LIN {X 0,Y 247.812,Z 545.239,A -85,B 0,C 180,E1 -18999.797,E2 -18999.797} C_VEL
LIN {X 0,Y 248.949,Z 540.408,A -85,B 0,C 180,E1 -19003.052,E2 -19003.052} C_VEL
LIN {X 0,Y 250.872,Z 533.939,A -85,B 0,C 180,E1 -19006.268,E2 -19006.268} C_VEL
LIN {X 0,Y 252.75,Z 526.871,A -85,B 0,C 180,E1 -19009.018,E2 -19009.018} C_VEL
LIN {X 0,Y 254.982,Z 519.187,A -85,B 0,C 180,E1 -19011.42,E2 -19011.42} C_VEL
LIN {X 0,Y 257.581,Z 510.12,A -85,B 0,C 180,E1 -19013.731,E2 -19013.731} C_VEL
LIN {X 0,Y 260.595,Z 499.136,A -85,B 0,C 180,E1 -19015.991,E2 -19015.991} C_VEL
LIN {X 0,Y 263.396,Z 487.928,A -85,B 0,C 180,E1 -19017.835,E2 -19017.835} C_VEL
LIN {X 0,Y 266.028,Z 475.354,A -85,B 0,C 180,E1 -19019.498,E2 -19019.498} C_VEL
LIN {X 0,Y 268.183,Z 463.582,A -85,B 0,C 180,E1 -19020.731,E2 -19020.731} C_VEL
LIN {X 0,Y 270.195,Z 450.492,A -85,B 0,C 180,E1 -19021.783,E2 -19021.783} C_VEL
LIN {X 0,Y 271.759,Z 437.252,A -85,B 0,C 180,E1 -19022.563,E2 -19022.563} C_VEL
LIN {X 0,Y 272.875,Z 422.735,A -85,B 0,C 180,E1 -19023.129,E2 -19023.129} C_VEL
LIN {X 0,Y 275.889,Z 350.665,A -85,B 0,C 180,E1 -19024.953,E2 -19024.953} C_VEL
LIN {X 0,Y 276.102,Z 341.819,A -85,B 0,C 180,E1 -19025.198,E2 -19025.198} C_VEL
LIN {X 0,Y 269.628,Z 326.55,A -85,B 0,C 180,E1 -19026.671,E2 -19026.671} C_VEL
LIN {X 0,Y 261.498,Z 310.016,A -85,B 0,C 180,E1 -19028.578,E2 -19028.578} C_VEL
LIN {X 0,Y 254.853,Z 298.261,A -85,B 0,C 180,E1 -19030.206,E2 -19030.206} C_VEL
LIN {X 0,Y 249.821,Z 289.724,A -85,B 0,C 180,E1 -19031.561,E2 -19031.561} C_VEL
LIN {X 0,Y 249.021,Z 287.115,A -85,B 0,C 180,E1 -19032.795,E2 -19032.795} C_VEL
LIN {X 0,Y 249.016,Z 287.053,A -85,B 0,C 180,E1 -19037.362,E2 -19037.362} C_VEL
LIN {X 0,Y 249.035,Z 287.087,A -85,B 0,C 180,E1 -19041.621,E2 -19041.621} C_VEL
LIN {X 0,Y 249.058,Z 287.032,A -85,B 0,C 180,E1 -19045.641,E2 -19045.641} C_VEL
LIN {X 0,Y 249.048,Z 287.064,A -85,B 0,C 180,E1 -19049.472,E2 -19049.472} C_VEL
LIN {X 0,Y 249.07,Z 287.07,A -85,B 0,C 180,E1 -19053.162,E2 -19053.162} C_VEL
LIN {X 0,Y 249.075,Z 287.086,A -85,B 0,C 180,E1 -19056.732,E2 -19056.732} C_VEL
LIN {X 0,Y 249.105,Z 287.065,A -85,B 0,C 180,E1 -19060.211,E2 -19060.211} C_VEL
LIN {X 0,Y 249.238,Z 287.051,A -85,B 0,C 180,E1 -19063.621,E2 -19063.621} C_VEL
LIN {X 0,Y 249.239,Z 287.062,A -85,B 0,C 180,E1 -19068.616,E2 -19068.616} C_VEL
LIN {X 0,Y 249.449,Z 287.016,A -85,B 0,C 180,E1 -19071.902,E2 -19071.902} C_VEL
LIN {X 0,Y 249.32,Z 287.04,A -85,B 0,C 180,E1 -19075.745,E2 -19075.745} C_VEL
LIN {X 0,Y 248.758,Z 287.101,A -85,B 0,C 180,E1 -19077.097,E2 -19077.097} C_VEL
LIN {X 0,Y 246.053,Z 287.448,A -85,B 0,C 180,E1 -19079.305,E2 -19079.305} C_VEL
LIN {X 0,Y 242.805,Z 287.856,A -85,B 0,C 180,E1 -19082.025,E2 -19082.025} C_VEL
LIN {X 0,Y 242.407,Z 287.894,A -85,B 0,C 180,E1 -19082.966,E2 -19082.966} C_VEL
LIN {X 0,Y 242.428,Z 287.91,A -85,B 0,C 180,E1 -19086.659,E2 -19086.659} C_VEL
LIN {X 0,Y 242.309,Z 287.903,A -85,B 0,C 180,E1 -19090.022,E2 -19090.022} C_VEL
LIN {X 0,Y 242.151,Z 287.932,A -85,B 0,C 180,E1 -19095.142,E2 -19095.142} C_VEL
LIN {X 0,Y 242.066,Z 287.954,A -85,B 0,C 180,E1 -19098.625,E2 -19098.625} C_VEL
LIN {X 0,Y 242.008,Z 287.945,A -85,B 0,C 180,E1 -19102.18,E2 -19102.18} C_VEL
LIN {X 0,Y 242.063,Z 287.951,A -85,B 0,C 180,E1 -19105.838,E2 -19105.838} C_VEL
LIN {X 0,Y 242.026,Z 287.962,A -85,B 0,C 180,E1 -19109.581,E2 -19109.581} C_VEL
LIN {X 0,Y 241.977,Z 287.91,A -85,B 0,C 180,E1 -19113.493,E2 -19113.493} C_VEL
LIN {X 0,Y 241.983,Z 287.952,A -85,B 0,C 180,E1 -19117.583,E2 -19117.583} C_VEL
LIN {X 0,Y 241.94,Z 287.97,A -85,B 0,C 180,E1 -19121.922,E2 -19121.922} C_VEL
LIN {X 0,Y 241.976,Z 288.026,A -85,B 0,C 180,E1 -19124.674,E2 -19124.674} C_VEL
LIN {X 0,Y 243.43,Z 292.652,A -85,B 0,C 180,E1 -19127.066,E2 -19127.066} C_VEL
LIN {X 0,Y 245.542,Z 296.633,A -85,B 0,C 180,E1 -19127.779,E2 -19127.779} C_VEL
LIN {X 0,Y 251.81,Z 307.211,A -85,B 0,C 180,E1 -19129.449,E2 -19129.449} C_VEL
LIN {X 0,Y 259.928,Z 322.862,A -85,B 0,C 180,E1 -19131.503,E2 -19131.503} C_VEL
LIN {X 0,Y 267.648,Z 340.131,A -85,B 0,C 180,E1 -19133.371,E2 -19133.371} C_VEL
LIN {X 0,Y 270.071,Z 346.299,A -85,B 0,C 180,E1 -19133.951,E2 -19133.951} C_VEL
LIN {X 0,Y 270.223,Z 349.656,A -85,B 0,C 180,E1 -19134.082,E2 -19134.082} C_VEL
LIN {X 0,Y 266.583,Z 431,A -85,B 0,C 180,E1 -19136.193,E2 -19136.193} C_VEL
LIN {X 0,Y 265.194,Z 445.012,A -85,B 0,C 180,E1 -19136.811,E2 -19136.811} C_VEL
LIN {X 0,Y 263.479,Z 457.894,A -85,B 0,C 180,E1 -19137.647,E2 -19137.647} C_VEL
LIN {X 0,Y 261.144,Z 471.147,A -85,B 0,C 180,E1 -19138.798,E2 -19138.798} C_VEL
LIN {X 0,Y 258.544,Z 483.922,A -85,B 0,C 180,E1 -19140.259,E2 -19140.259} C_VEL
LIN {X 0,Y 255.96,Z 495.088,A -85,B 0,C 180,E1 -19141.867,E2 -19141.867} C_VEL
LIN {X 0,Y 253.272,Z 505.213,A -85,B 0,C 180,E1 -19143.643,E2 -19143.643} C_VEL
LIN {X 0,Y 250.226,Z 515.932,A -85,B 0,C 180,E1 -19145.968,E2 -19145.968} C_VEL
LIN {X 0,Y 247.534,Z 524.782,A -85,B 0,C 180,E1 -19148.341,E2 -19148.341} C_VEL
LIN {X 0,Y 245.329,Z 532.305,A -85,B 0,C 180,E1 -19150.827,E2 -19150.827} C_VEL
LIN {X 0,Y 243.603,Z 538.288,A -85,B 0,C 180,E1 -19153.232,E2 -19153.232} C_VEL
LIN {X 0,Y 242.131,Z 543.376,A -85,B 0,C 180,E1 -19155.717,E2 -19155.717} C_VEL
LIN {X 0,Y 240.791,Z 548.626,A -85,B 0,C 180,E1 -19159.064,E2 -19159.064} C_VEL
LIN {X 0,Y 240.204,Z 551.568,A -85,B 0,C 180,E1 -19161.588,E2 -19161.588} C_VEL
LIN {X 0,Y 239.8,Z 554.259,A -85,B 0,C 180,E1 -19164.956,E2 -19164.956} C_VEL
LIN {X 0,Y 239.768,Z 555.59,A -85,B 0,C 180,E1 -19168.32,E2 -19168.32} C_VEL
LIN {X 0,Y 239.802,Z 555.753,A -85,B 0,C 180,E1 -19170,E2 -19170} C_VEL
LIN {X 0,Y 239.727,Z 555.077,A -85,B 0,C 180,E1 -19173.361,E2 -19173.361} C_VEL
LIN {X 0,Y 239.955,Z 553.058,A -85,B 0,C 180,E1 -19176.728,E2 -19176.728} C_VEL
LIN {X 0,Y 240.584,Z 549.648,A -85,B 0,C 180,E1 -19180.094,E2 -19180.094} C_VEL
LIN {X 0,Y 241.671,Z 544.743,A -85,B 0,C 180,E1 -19183.453,E2 -19183.453} C_VEL
LIN {X 0,Y 243.115,Z 540.017,A -85,B 0,C 180,E1 -19185.94,E2 -19185.94} C_VEL
LIN {X 0,Y 244.834,Z 533.55,A -85,B 0,C 180,E1 -19188.689,E2 -19188.689} C_VEL
LIN {X 0,Y 247.121,Z 526.01,A -85,B 0,C 180,E1 -19191.26,E2 -19191.26} C_VEL
LIN {X 0,Y 249.716,Z 517.407,A -85,B 0,C 180,E1 -19193.643,E2 -19193.643} C_VEL
LIN {X 0,Y 252.713,Z 506.979,A -85,B 0,C 180,E1 -19195.976,E2 -19195.976} C_VEL
LIN {X 0,Y 255.58,Z 496.491,A -85,B 0,C 180,E1 -19197.87,E2 -19197.87} C_VEL
LIN {X 0,Y 258.224,Z 485.076,A -85,B 0,C 180,E1 -19199.557,E2 -19199.557} C_VEL
LIN {X 0,Y 260.813,Z 472.57,A -85,B 0,C 180,E1 -19201.02,E2 -19201.02} C_VEL
LIN {X 0,Y 263.278,Z 458.571,A -85,B 0,C 180,E1 -19202.268,E2 -19202.268} C_VEL
LIN {X 0,Y 265.197,Z 444.403,A -85,B 0,C 180,E1 -19203.189,E2 -19203.189} C_VEL
LIN {X 0,Y 266.527,Z 431.14,A -85,B 0,C 180,E1 -19203.764,E2 -19203.764} C_VEL
LIN {X 0,Y 270.16,Z 347.755,A -85,B 0,C 180,E1 -19205.943,E2 -19205.943} C_VEL
LIN {X 0,Y 269.356,Z 344.393,A -85,B 0,C 180,E1 -19206.175,E2 -19206.175} C_VEL
LIN {X 0,Y 261.649,Z 326.639,A -85,B 0,C 180,E1 -19208.018,E2 -19208.018} C_VEL
LIN {X 0,Y 255.334,Z 313.91,A -85,B 0,C 180,E1 -19209.584,E2 -19209.584} C_VEL
LIN {X 0,Y 248.605,Z 301.75,A -85,B 0,C 180,E1 -19211.33,E2 -19211.33} C_VEL
LIN {X 0,Y 243.519,Z 293.077,A -85,B 0,C 180,E1 -19212.766,E2 -19212.766} C_VEL
LIN {X 0,Y 242.068,Z 288.569,A -85,B 0,C 180,E1 -19214.876,E2 -19214.876} C_VEL
LIN {X 0,Y 241.951,Z 287.996,A -85,B 0,C 180,E1 -19215.327,E2 -19215.327} C_VEL
LIN {X 0,Y 241.929,Z 287.963,A -85,B 0,C 180,E1 -19219.05,E2 -19219.05} C_VEL
LIN {X 0,Y 241.984,Z 287.949,A -85,B 0,C 180,E1 -19222.417,E2 -19222.417} C_VEL
LIN {X 0,Y 241.977,Z 287.91,A -85,B 0,C 180,E1 -19226.507,E2 -19226.507} C_VEL
LIN {X 0,Y 242.034,Z 287.96,A -85,B 0,C 180,E1 -19230.587,E2 -19230.587} C_VEL
LIN {X 0,Y 242.064,Z 287.951,A -85,B 0,C 180,E1 -19234.183,E2 -19234.183} C_VEL
LIN {X 0,Y 242.049,Z 287.94,A -85,B 0,C 180,E1 -19238.297,E2 -19238.297} C_VEL
LIN {X 0,Y 242.16,Z 287.924,A -85,B 0,C 180,E1 -19243.278,E2 -19243.278} C_VEL
LIN {X 0,Y 242.181,Z 287.927,A -85,B 0,C 180,E1 -19248.28,E2 -19248.28} C_VEL
LIN {X 0,Y 242.423,Z 287.905,A -85,B 0,C 180,E1 -19251.666,E2 -19251.666} C_VEL
LIN {X 0,Y 242.253,Z 287.912,A -85,B 0,C 180,E1 -19255.007,E2 -19255.007} C_VEL
LIN {X 0,Y 242.631,Z 287.883,A -85,B 0,C 180,E1 -19258.34,E2 -19258.34} C_VEL
LIN {X 0,Y 242.632,Z 287.863,A -85,B 0,C 180,E1 -19261.66,E2 -19261.66} C_VEL
LIN {X 0,Y 242.417,Z 287.908,A -85,B 0,C 180,E1 -19266.682,E2 -19266.682} C_VEL
LIN {X 0,Y 242.263,Z 287.914,A -85,B 0,C 180,E1 -19270.024,E2 -19270.024} C_VEL
LIN {X 0,Y 242.159,Z 287.923,A -85,B 0,C 180,E1 -19275.141,E2 -19275.141} C_VEL
LIN {X 0,Y 242.069,Z 287.955,A -85,B 0,C 180,E1 -19278.625,E2 -19278.625} C_VEL
LIN {X 0,Y 242.01,Z 287.951,A -85,B 0,C 180,E1 -19282.18,E2 -19282.18} C_VEL
LIN {X 0,Y 242.064,Z 287.94,A -85,B 0,C 180,E1 -19285.839,E2 -19285.839} C_VEL
LIN {X 0,Y 242.028,Z 287.959,A -85,B 0,C 180,E1 -19289.581,E2 -19289.581} C_VEL
LIN {X 0,Y 241.989,Z 287.902,A -85,B 0,C 180,E1 -19293.492,E2 -19293.492} C_VEL
LIN {X 0,Y 242.002,Z 287.967,A -85,B 0,C 180,E1 -19297.58,E2 -19297.58} C_VEL
LIN {X 0,Y 241.942,Z 287.925,A -85,B 0,C 180,E1 -19301.922,E2 -19301.922} C_VEL
LIN {X 0,Y 241.972,Z 288.119,A -85,B 0,C 180,E1 -19306.277,E2 -19306.277} C_VEL
LIN {X 0,Y 242.426,Z 289.737,A -85,B 0,C 180,E1 -19307.011,E2 -19307.011} C_VEL
LIN {X 0,Y 246.633,Z 296.686,A -85,B 0,C 180,E1 -19308.25,E2 -19308.25} C_VEL
LIN {X 0,Y 253.42,Z 308.137,A -85,B 0,C 180,E1 -19310.026,E2 -19310.026} C_VEL
LIN {X 0,Y 260.799,Z 322.351,A -85,B 0,C 180,E1 -19311.866,E2 -19311.866} C_VEL
LIN {X 0,Y 268.081,Z 338.456,A -85,B 0,C 180,E1 -19313.609,E2 -19313.609} C_VEL
LIN {X 0,Y 270.243,Z 343.753,A -85,B 0,C 180,E1 -19314.118,E2 -19314.118} C_VEL
LIN {X 0,Y 267.245,Z 415.04,A -85,B 0,C 180,E1 -19315.949,E2 -19315.949} C_VEL
LIN {X 0,Y 266.306,Z 431.164,A -85,B 0,C 180,E1 -19316.458,E2 -19316.458} C_VEL
LIN {X 0,Y 264.801,Z 444.962,A -85,B 0,C 180,E1 -19317.152,E2 -19317.152} C_VEL
LIN {X 0,Y 262.871,Z 458.452,A -85,B 0,C 180,E1 -19318.128,E2 -19318.128} C_VEL
LIN {X 0,Y 260.555,Z 471.491,A -85,B 0,C 180,E1 -19319.396,E2 -19319.396} C_VEL
LIN {X 0,Y 258.137,Z 483.353,A -85,B 0,C 180,E1 -19320.879,E2 -19320.879} C_VEL
LIN {X 0,Y 255.451,Z 494.306,A -85,B 0,C 180,E1 -19322.56,E2 -19322.56} C_VEL
LIN {X 0,Y 252.662,Z 504.432,A -85,B 0,C 180,E1 -19324.46,E2 -19324.46} C_VEL
LIN {X 0,Y 249.805,Z 514.482,A -85,B 0,C 180,E1 -19326.805,E2 -19326.805} C_VEL
LIN {X 0,Y 247.208,Z 522.827,A -85,B 0,C 180,E1 -19329.184,E2 -19329.184} C_VEL
LIN {X 0,Y 244.883,Z 530.796,A -85,B 0,C 180,E1 -19332.03,E2 -19332.03} C_VEL
LIN {X 0,Y 243.509,Z 535.534,A -85,B 0,C 180,E1 -19334.087,E2 -19334.087} C_VEL
LIN {X 0,Y 242.019,Z 540.257,A -85,B 0,C 180,E1 -19336.567,E2 -19336.567} C_VEL
LIN {X 0,Y 240.792,Z 545.147,A -85,B 0,C 180,E1 -19339.914,E2 -19339.914} C_VEL
LIN {X 0,Y 240.102,Z 548.549,A -85,B 0,C 180,E1 -19343.276,E2 -19343.276} C_VEL
LIN {X 0,Y 239.799,Z 550.567,A -85,B 0,C 180,E1 -19346.64,E2 -19346.64} C_VEL
LIN {X 0,Y 239.806,Z 551.254,A -85,B 0,C 180,E1 -19350,E2 -19350} C_VEL
LIN {X 0,Y 239.8,Z 550.623,A -85,B 0,C 180,E1 -19353.36,E2 -19353.36} C_VEL
LIN {X 0,Y 240.1,Z 548.655,A -85,B 0,C 180,E1 -19356.724,E2 -19356.724} C_VEL
LIN {X 0,Y 240.779,Z 545.305,A -85,B 0,C 180,E1 -19360.086,E2 -19360.086} C_VEL
LIN {X 0,Y 241.996,Z 540.474,A -85,B 0,C 180,E1 -19363.434,E2 -19363.434} C_VEL
LIN {X 0,Y 244.043,Z 534.004,A -85,B 0,C 180,E1 -19366.737,E2 -19366.737} C_VEL
LIN {X 0,Y 245.873,Z 527.398,A -85,B 0,C 180,E1 -19369.392,E2 -19369.392} C_VEL
LIN {X 0,Y 248.348,Z 519.252,A -85,B 0,C 180,E1 -19372.021,E2 -19372.021} C_VEL
LIN {X 0,Y 251.081,Z 510.184,A -85,B 0,C 180,E1 -19374.384,E2 -19374.384} C_VEL
LIN {X 0,Y 254.217,Z 499.199,A -85,B 0,C 180,E1 -19376.694,E2 -19376.694} C_VEL
LIN {X 0,Y 257.139,Z 487.991,A -85,B 0,C 180,E1 -19378.574,E2 -19378.574} C_VEL
LIN {X 0,Y 259.832,Z 475.594,A -85,B 0,C 180,E1 -19380.248,E2 -19380.248} C_VEL
LIN {X 0,Y 262.119,Z 463.641,A -85,B 0,C 180,E1 -19381.522,E2 -19381.522} C_VEL
LIN {X 0,Y 264.189,Z 450.55,A -85,B 0,C 180,E1 -19382.594,E2 -19382.594} C_VEL
LIN {X 0,Y 265.816,Z 437.306,A -85,B 0,C 180,E1 -19383.384,E2 -19383.384} C_VEL
LIN {X 0,Y 266.931,Z 423.228,A -85,B 0,C 180,E1 -19383.948,E2 -19383.948} C_VEL
LIN {X 0,Y 269.97,Z 354.319,A -85,B 0,C 180,E1 -19385.72,E2 -19385.72} C_VEL
LIN {X 0,Y 270.252,Z 343.785,A -85,B 0,C 180,E1 -19386.015,E2 -19386.015} C_VEL
LIN {X 0,Y 263.395,Z 327.749,A -85,B 0,C 180,E1 -19387.648,E2 -19387.648} C_VEL
LIN {X 0,Y 255.001,Z 310.963,A -85,B 0,C 180,E1 -19389.72,E2 -19389.72} C_VEL
LIN {X 0,Y 247.137,Z 297.487,A -85,B 0,C 180,E1 -19391.767,E2 -19391.767} C_VEL
LIN {X 0,Y 242.501,Z 289.81,A -85,B 0,C 180,E1 -19393.116,E2 -19393.116} C_VEL
LIN {X 0,Y 241.996,Z 288.031,A -85,B 0,C 180,E1 -19393.968,E2 -19393.968} C_VEL
LIN {X 0,Y 241.942,Z 287.927,A -85,B 0,C 180,E1 -19398.078,E2 -19398.078} C_VEL
LIN {X 0,Y 242,Z 287.971,A -85,B 0,C 180,E1 -19402.42,E2 -19402.42} C_VEL
LIN {X 0,Y 241.988,Z 287.906,A -85,B 0,C 180,E1 -19406.508,E2 -19406.508} C_VEL
LIN {X 0,Y 242.033,Z 287.961,A -85,B 0,C 180,E1 -19410.586,E2 -19410.586} C_VEL
LIN {X 0,Y 242.064,Z 287.94,A -85,B 0,C 180,E1 -19414.182,E2 -19414.182} C_VEL
LIN {X 0,Y 242.049,Z 287.943,A -85,B 0,C 180,E1 -19418.297,E2 -19418.297} C_VEL
LIN {X 0,Y 242.159,Z 287.938,A -85,B 0,C 180,E1 -19423.278,E2 -19423.278} C_VEL
LIN {X 0,Y 242.175,Z 287.944,A -85,B 0,C 180,E1 -19428.279,E2 -19428.279} C_VEL
LIN {X 0,Y 242.395,Z 287.892,A -85,B 0,C 180,E1 -19431.664,E2 -19431.664} C_VEL
LIN {X 0,Y 242.253,Z 287.932,A -85,B 0,C 180,E1 -19435.007,E2 -19435.007} C_VEL
LIN {X 0,Y 242.631,Z 287.862,A -85,B 0,C 180,E1 -19438.34,E2 -19438.34} C_VEL
LIN {X 0,Y 242.631,Z 287.883,A -85,B 0,C 180,E1 -19441.66,E2 -19441.66} C_VEL
LIN {X 0,Y 242.407,Z 287.894,A -85,B 0,C 180,E1 -19442.966,E2 -19442.966} C_VEL
LIN {X 0,Y 241.647,Z 287.99,A -85,B 0,C 180,E1 -19444.352,E2 -19444.352} C_VEL
LIN {X 0,Y 238.824,Z 288.358,A -85,B 0,C 180,E1 -19446.615,E2 -19446.615} C_VEL
LIN {X 0,Y 235.613,Z 288.742,A -85,B 0,C 180,E1 -19449.405,E2 -19449.405} C_VEL
LIN {X 0,Y 235.228,Z 288.784,A -85,B 0,C 180,E1 -19450.37,E2 -19450.37} C_VEL
LIN {X 0,Y 235.102,Z 288.805,A -85,B 0,C 180,E1 -19455.607,E2 -19455.607} C_VEL
LIN {X 0,Y 235.003,Z 288.837,A -85,B 0,C 180,E1 -19459.206,E2 -19459.206} C_VEL
LIN {X 0,Y 234.957,Z 288.825,A -85,B 0,C 180,E1 -19462.883,E2 -19462.883} C_VEL
LIN {X 0,Y 234.966,Z 288.826,A -85,B 0,C 180,E1 -19466.658,E2 -19466.658} C_VEL
LIN {X 0,Y 234.928,Z 288.843,A -85,B 0,C 180,E1 -19470.568,E2 -19470.568} C_VEL
LIN {X 0,Y 234.923,Z 288.784,A -85,B 0,C 180,E1 -19474.639,E2 -19474.639} C_VEL
LIN {X 0,Y 234.939,Z 288.843,A -85,B 0,C 180,E1 -19478.945,E2 -19478.945} C_VEL
LIN {X 0,Y 234.92,Z 289.02,A -85,B 0,C 180,E1 -19483.478,E2 -19483.478} C_VEL
LIN {X 0,Y 236.157,Z 292.844,A -85,B 0,C 180,E1 -19485.459,E2 -19485.459} C_VEL
LIN {X 0,Y 240.318,Z 299.833,A -85,B 0,C 180,E1 -19486.769,E2 -19486.769} C_VEL
LIN {X 0,Y 245.548,Z 308.586,A -85,B 0,C 180,E1 -19488.241,E2 -19488.241} C_VEL
LIN {X 0,Y 252.424,Z 321.534,A -85,B 0,C 180,E1 -19490.09,E2 -19490.09} C_VEL
LIN {X 0,Y 259.854,Z 337.413,A -85,B 0,C 180,E1 -19491.992,E2 -19491.992} C_VEL
LIN {X 0,Y 264.51,Z 348.754,A -85,B 0,C 180,E1 -19493.152,E2 -19493.152} C_VEL
LIN {X 0,Y 260.793,Z 430.168,A -85,B 0,C 180,E1 -19495.298,E2 -19495.298} C_VEL
LIN {X 0,Y 259.399,Z 444.192,A -85,B 0,C 180,E1 -19495.911,E2 -19495.911} C_VEL
LIN {X 0,Y 257.699,Z 456.701,A -85,B 0,C 180,E1 -19496.713,E2 -19496.713} C_VEL
LIN {X 0,Y 255.465,Z 469.318,A -85,B 0,C 180,E1 -19497.791,E2 -19497.791} C_VEL
LIN {X 0,Y 252.712,Z 482.433,A -85,B 0,C 180,E1 -19499.269,E2 -19499.269} C_VEL
LIN {X 0,Y 250.095,Z 493.748,A -85,B 0,C 180,E1 -19500.896,E2 -19500.896} C_VEL
LIN {X 0,Y 246.917,Z 505.149,A -85,B 0,C 180,E1 -19502.91,E2 -19502.91} C_VEL
LIN {X 0,Y 244.201,Z 514.238,A -85,B 0,C 180,E1 -19504.882,E2 -19504.882} C_VEL
LIN {X 0,Y 241.378,Z 523.362,A -85,B 0,C 180,E1 -19507.308,E2 -19507.308} C_VEL
LIN {X 0,Y 239.004,Z 530.966,A -85,B 0,C 180,E1 -19509.788,E2 -19509.788} C_VEL
LIN {X 0,Y 236.777,Z 538.223,A -85,B 0,C 180,E1 -19512.734,E2 -19512.734} C_VEL
LIN {X 0,Y 235.233,Z 543.31,A -85,B 0,C 180,E1 -19515.289,E2 -19515.289} C_VEL
LIN {X 0,Y 233.78,Z 548.56,A -85,B 0,C 180,E1 -19518.732,E2 -19518.732} C_VEL
LIN {X 0,Y 233.17,Z 551.502,A -85,B 0,C 180,E1 -19521.332,E2 -19521.332} C_VEL
LIN {X 0,Y 232.73,Z 554.193,A -85,B 0,C 180,E1 -19524.802,E2 -19524.802} C_VEL
LIN {X 0,Y 232.665,Z 555.523,A -85,B 0,C 180,E1 -19528.269,E2 -19528.269} C_VEL
LIN {X 0,Y 232.717,Z 555.687,A -85,B 0,C 180,E1 -19530,E2 -19530} C_VEL
LIN {X 0,Y 232.639,Z 555.01,A -85,B 0,C 180,E1 -19533.464,E2 -19533.464} C_VEL
LIN {X 0,Y 232.891,Z 552.991,A -85,B 0,C 180,E1 -19536.933,E2 -19536.933} C_VEL
LIN {X 0,Y 233.553,Z 549.58,A -85,B 0,C 180,E1 -19540.402,E2 -19540.402} C_VEL
LIN {X 0,Y 234.74,Z 544.675,A -85,B 0,C 180,E1 -19543.858,E2 -19543.858} C_VEL
LIN {X 0,Y 236.255,Z 539.948,A -85,B 0,C 180,E1 -19546.415,E2 -19546.415} C_VEL
LIN {X 0,Y 238.18,Z 533.206,A -85,B 0,C 180,E1 -19549.342,E2 -19549.342} C_VEL
LIN {X 0,Y 240.901,Z 524.585,A -85,B 0,C 180,E1 -19552.287,E2 -19552.287} C_VEL
LIN {X 0,Y 243.723,Z 515.709,A -85,B 0,C 180,E1 -19554.716,E2 -19554.716} C_VEL
LIN {X 0,Y 246.336,Z 506.909,A -85,B 0,C 180,E1 -19556.701,E2 -19556.701} C_VEL
LIN {X 0,Y 249.305,Z 496.421,A -85,B 0,C 180,E1 -19558.635,E2 -19558.635} C_VEL
LIN {X 0,Y 252.043,Z 485.005,A -85,B 0,C 180,E1 -19560.357,E2 -19560.357} C_VEL
LIN {X 0,Y 254.755,Z 472.498,A -85,B 0,C 180,E1 -19561.843,E2 -19561.843} C_VEL
LIN {X 0,Y 257.317,Z 458.498,A -85,B 0,C 180,E1 -19563.11,E2 -19563.11} C_VEL
LIN {X 0,Y 259.29,Z 444.328,A -85,B 0,C 180,E1 -19564.047,E2 -19564.047} C_VEL
LIN {X 0,Y 260.655,Z 431.188,A -85,B 0,C 180,E1 -19564.624,E2 -19564.624} C_VEL
LIN {X 0,Y 263.847,Z 360.851,A -85,B 0,C 180,E1 -19566.505,E2 -19566.505} C_VEL
LIN {X 0,Y 264.347,Z 348.464,A -85,B 0,C 180,E1 -19566.835,E2 -19566.835} C_VEL
LIN {X 0,Y 256.887,Z 330.881,A -85,B 0,C 180,E1 -19568.702,E2 -19568.702} C_VEL
LIN {X 0,Y 250.242,Z 317.359,A -85,B 0,C 180,E1 -19570.424,E2 -19570.424} C_VEL
LIN {X 0,Y 244.162,Z 306.242,A -85,B 0,C 180,E1 -19572.077,E2 -19572.077} C_VEL
LIN {X 0,Y 238.387,Z 296.737,A -85,B 0,C 180,E1 -19573.725,E2 -19573.725} C_VEL
LIN {X 0,Y 236.013,Z 292.565,A -85,B 0,C 180,E1 -19574.567,E2 -19574.567} C_VEL
LIN {X 0,Y 234.902,Z 288.881,A -85,B 0,C 180,E1 -19576.583,E2 -19576.583} C_VEL
LIN {X 0,Y 234.916,Z 288.848,A -85,B 0,C 180,E1 -19581.078,E2 -19581.078} C_VEL
LIN {X 0,Y 234.924,Z 288.783,A -85,B 0,C 180,E1 -19585.361,E2 -19585.361} C_VEL
LIN {X 0,Y 234.928,Z 288.844,A -85,B 0,C 180,E1 -19589.432,E2 -19589.432} C_VEL
LIN {X 0,Y 234.991,Z 288.828,A -85,B 0,C 180,E1 -19593.793,E2 -19593.793} C_VEL
LIN {X 0,Y 235.008,Z 288.822,A -85,B 0,C 180,E1 -19598.97,E2 -19598.97} C_VEL
LIN {X 0,Y 235.092,Z 288.804,A -85,B 0,C 180,E1 -19603.06,E2 -19603.06} C_VEL
LIN {X 0,Y 235.141,Z 288.808,A -85,B 0,C 180,E1 -19607.924,E2 -19607.924} C_VEL
LIN {X 0,Y 235.373,Z 288.78,A -85,B 0,C 180,E1 -19611.414,E2 -19611.414} C_VEL
LIN {X 0,Y 235.399,Z 288.788,A -85,B 0,C 180,E1 -19613.141,E2 -19613.141} C_VEL
LIN {X 0,Y 235.591,Z 288.758,A -85,B 0,C 180,E1 -19618.291,E2 -19618.291} C_VEL
LIN {X 0,Y 235.591,Z 288.739,A -85,B 0,C 180,E1 -19621.71,E2 -19621.71} C_VEL
LIN {X 0,Y 235.369,Z 288.783,A -85,B 0,C 180,E1 -19626.86,E2 -19626.86} C_VEL
LIN {X 0,Y 235.21,Z 288.795,A -85,B 0,C 180,E1 -19630.328,E2 -19630.328} C_VEL
LIN {X 0,Y 235.108,Z 288.802,A -85,B 0,C 180,E1 -19635.607,E2 -19635.607} C_VEL
LIN {X 0,Y 235.005,Z 288.828,A -85,B 0,C 180,E1 -19639.206,E2 -19639.206} C_VEL
LIN {X 0,Y 234.958,Z 288.839,A -85,B 0,C 180,E1 -19642.883,E2 -19642.883} C_VEL
LIN {X 0,Y 234.967,Z 288.823,A -85,B 0,C 180,E1 -19646.658,E2 -19646.658} C_VEL
LIN {X 0,Y 234.929,Z 288.818,A -85,B 0,C 180,E1 -19650.568,E2 -19650.568} C_VEL
LIN {X 0,Y 234.958,Z 288.783,A -85,B 0,C 180,E1 -19654.634,E2 -19654.634} C_VEL
LIN {X 0,Y 234.94,Z 288.824,A -85,B 0,C 180,E1 -19658.945,E2 -19658.945} C_VEL
LIN {X 0,Y 234.888,Z 288.819,A -85,B 0,C 180,E1 -19663.486,E2 -19663.486} C_VEL
LIN {X 0,Y 234.924,Z 289.112,A -85,B 0,C 180,E1 -19665.035,E2 -19665.035} C_VEL
LIN {X 0,Y 235.122,Z 289.995,A -85,B 0,C 180,E1 -19665.35,E2 -19665.35} C_VEL
LIN {X 0,Y 236.786,Z 292.857,A -85,B 0,C 180,E1 -19665.921,E2 -19665.921} C_VEL
LIN {X 0,Y 241.532,Z 299.933,A -85,B 0,C 180,E1 -19667.286,E2 -19667.286} C_VEL
LIN {X 0,Y 249.277,Z 313.414,A -85,B 0,C 180,E1 -19669.417,E2 -19669.417} C_VEL
LIN {X 0,Y 255.861,Z 326.217,A -85,B 0,C 180,E1 -19671.127,E2 -19671.127} C_VEL
LIN {X 0,Y 263.09,Z 342.441,A -85,B 0,C 180,E1 -19672.935,E2 -19672.935} C_VEL
LIN {X 0,Y 264.524,Z 346.43,A -85,B 0,C 180,E1 -19673.303,E2 -19673.303} C_VEL
LIN {X 0,Y 260.778,Z 426.423,A -85,B 0,C 180,E1 -19675.401,E2 -19675.401} C_VEL
LIN {X 0,Y 259.328,Z 441.233,A -85,B 0,C 180,E1 -19676.076,E2 -19676.076} C_VEL
LIN {X 0,Y 257.383,Z 455.146,A -85,B 0,C 180,E1 -19677.017,E2 -19677.017} C_VEL
LIN {X 0,Y 255.125,Z 468.094,A -85,B 0,C 180,E1 -19678.208,E2 -19678.208} C_VEL
LIN {X 0,Y 252.568,Z 480.565,A -85,B 0,C 180,E1 -19679.7,E2 -19679.7} C_VEL
LIN {X 0,Y 249.776,Z 492.082,A -85,B 0,C 180,E1 -19681.424,E2 -19681.424} C_VEL
LIN {X 0,Y 246.809,Z 502.585,A -85,B 0,C 180,E1 -19683.354,E2 -19683.354} C_VEL
LIN {X 0,Y 243.731,Z 513.014,A -85,B 0,C 180,E1 -19685.739,E2 -19685.739} C_VEL
LIN {X 0,Y 240.958,Z 521.616,A -85,B 0,C 180,E1 -19688.169,E2 -19688.169} C_VEL
LIN {X 0,Y 238.407,Z 529.858,A -85,B 0,C 180,E1 -19691.079,E2 -19691.079} C_VEL
LIN {X 0,Y 236.665,Z 535.603,A -85,B 0,C 180,E1 -19693.614,E2 -19693.614} C_VEL
LIN {X 0,Y 235.083,Z 540.325,A -85,B 0,C 180,E1 -19696.163,E2 -19696.163} C_VEL
LIN {X 0,Y 233.78,Z 545.215,A -85,B 0,C 180,E1 -19699.609,E2 -19699.609} C_VEL
LIN {X 0,Y 233.052,Z 548.616,A -85,B 0,C 180,E1 -19703.072,E2 -19703.072} C_VEL
LIN {X 0,Y 232.712,Z 550.634,A -85,B 0,C 180,E1 -19706.537,E2 -19706.537} C_VEL
LIN {X 0,Y 232.721,Z 551.321,A -85,B 0,C 180,E1 -19710,E2 -19710} C_VEL
LIN {X 0,Y 232.713,Z 550.689,A -85,B 0,C 180,E1 -19713.463,E2 -19713.463} C_VEL
LIN {X 0,Y 233.049,Z 548.721,A -85,B 0,C 180,E1 -19716.928,E2 -19716.928} C_VEL
LIN {X 0,Y 233.763,Z 545.371,A -85,B 0,C 180,E1 -19720.392,E2 -19720.392} C_VEL
LIN {X 0,Y 235.06,Z 540.54,A -85,B 0,C 180,E1 -19723.838,E2 -19723.838} C_VEL
LIN {X 0,Y 237.207,Z 534.069,A -85,B 0,C 180,E1 -19727.234,E2 -19727.234} C_VEL
LIN {X 0,Y 239.352,Z 526.823,A -85,B 0,C 180,E1 -19730.2,E2 -19730.2} C_VEL
LIN {X 0,Y 242.206,Z 517.953,A -85,B 0,C 180,E1 -19733.061,E2 -19733.061} C_VEL
LIN {X 0,Y 245.134,Z 508.586,A -85,B 0,C 180,E1 -19735.47,E2 -19735.47} C_VEL
LIN {X 0,Y 248.167,Z 498.213,A -85,B 0,C 180,E1 -19737.628,E2 -19737.628} C_VEL
LIN {X 0,Y 251.216,Z 486.846,A -85,B 0,C 180,E1 -19739.527,E2 -19739.527} C_VEL
LIN {X 0,Y 253.944,Z 474.387,A -85,B 0,C 180,E1 -19741.212,E2 -19741.212} C_VEL
LIN {X 0,Y 256.43,Z 461.716,A -85,B 0,C 180,E1 -19742.537,E2 -19742.537} C_VEL
LIN {X 0,Y 258.584,Z 448.008,A -85,B 0,C 180,E1 -19743.625,E2 -19743.625} C_VEL
LIN {X 0,Y 260.285,Z 433.7,A -85,B 0,C 180,E1 -19744.425,E2 -19744.425} C_VEL
LIN {X 0,Y 261.265,Z 420.071,A -85,B 0,C 180,E1 -19744.914,E2 -19744.914} C_VEL
LIN {X 0,Y 264.419,Z 349.554,A -85,B 0,C 180,E1 -19746.749,E2 -19746.749} C_VEL
LIN {X 0,Y 264.411,Z 345.633,A -85,B 0,C 180,E1 -19746.881,E2 -19746.881} C_VEL
LIN {X 0,Y 257.553,Z 329.735,A -85,B 0,C 180,E1 -19748.59,E2 -19748.59} C_VEL
LIN {X 0,Y 249.855,Z 314.362,A -85,B 0,C 180,E1 -19750.583,E2 -19750.583} C_VEL
LIN {X 0,Y 242.786,Z 302.148,A -85,B 0,C 180,E1 -19752.508,E2 -19752.508} C_VEL
LIN {X 0,Y 237.087,Z 293.091,A -85,B 0,C 180,E1 -19754.159,E2 -19754.159} C_VEL
LIN {X 0,Y 235.348,Z 290.564,A -85,B 0,C 180,E1 -19754.705,E2 -19754.705} C_VEL
LIN {X 0,Y 234.959,Z 289.153,A -85,B 0,C 180,E1 -19755.095,E2 -19755.095} C_VEL
LIN {X 0,Y 234.888,Z 288.823,A -85,B 0,C 180,E1 -19756.514,E2 -19756.514} C_VEL
LIN {X 0,Y 234.953,Z 288.823,A -85,B 0,C 180,E1 -19761.085,E2 -19761.085} C_VEL
LIN {X 0,Y 234.958,Z 288.788,A -85,B 0,C 180,E1 -19765.366,E2 -19765.366} C_VEL
LIN {X 0,Y 234.966,Z 288.832,A -85,B 0,C 180,E1 -19770.157,E2 -19770.157} C_VEL
LIN {X 0,Y 234.991,Z 288.821,A -85,B 0,C 180,E1 -19773.793,E2 -19773.793} C_VEL
LIN {X 0,Y 235.007,Z 288.816,A -85,B 0,C 180,E1 -19778.969,E2 -19778.969} C_VEL
LIN {X 0,Y 235.092,Z 288.82,A -85,B 0,C 180,E1 -19783.059,E2 -19783.059} C_VEL
LIN {X 0,Y 235.109,Z 288.823,A -85,B 0,C 180,E1 -19787.922,E2 -19787.922} C_VEL
LIN {X 0,Y 235.326,Z 288.772,A -85,B 0,C 180,E1 -19791.412,E2 -19791.412} C_VEL
LIN {X 0,Y 235.369,Z 288.782,A -85,B 0,C 180,E1 -19793.14,E2 -19793.14} C_VEL
LIN {X 0,Y 235.591,Z 288.739,A -85,B 0,C 180,E1 -19798.29,E2 -19798.29} C_VEL
LIN {X 0,Y 235.591,Z 288.759,A -85,B 0,C 180,E1 -19801.709,E2 -19801.709} C_VEL
LIN {X 0,Y 235.399,Z 288.788,A -85,B 0,C 180,E1 -19806.859,E2 -19806.859} C_VEL
LIN {X 0,Y 235.228,Z 288.784,A -85,B 0,C 180,E1 -19810.37,E2 -19810.37} C_VEL
LIN {X 0,Y 234.467,Z 288.891,A -85,B 0,C 180,E1 -19811.796,E2 -19811.796} C_VEL
LIN {X 0,Y 231.611,Z 289.257,A -85,B 0,C 180,E1 -19814.125,E2 -19814.125} C_VEL
LIN {X 0,Y 228.372,Z 289.653,A -85,B 0,C 180,E1 -19816.998,E2 -19816.998} C_VEL
LIN {X 0,Y 227.994,Z 289.697,A -85,B 0,C 180,E1 -19817.993,E2 -19817.993} C_VEL
LIN {X 0,Y 227.926,Z 289.698,A -85,B 0,C 180,E1 -19822.329,E2 -19822.329} C_VEL
LIN {X 0,Y 227.939,Z 289.701,A -85,B 0,C 180,E1 -19826.603,E2 -19826.603} C_VEL
LIN {X 0,Y 227.905,Z 289.721,A -85,B 0,C 180,E1 -19830.296,E2 -19830.296} C_VEL
LIN {X 0,Y 227.873,Z 289.663,A -85,B 0,C 180,E1 -19833.721,E2 -19833.721} C_VEL
LIN {X 0,Y 227.841,Z 289.723,A -85,B 0,C 180,E1 -19838.092,E2 -19838.092} C_VEL
LIN {X 0,Y 227.876,Z 289.933,A -85,B 0,C 180,E1 -19842.09,E2 -19842.09} C_VEL
LIN {X 0,Y 228.816,Z 292.87,A -85,B 0,C 180,E1 -19843.64,E2 -19843.64} C_VEL
LIN {X 0,Y 231.677,Z 297.405,A -85,B 0,C 180,E1 -19844.624,E2 -19844.624} C_VEL
LIN {X 0,Y 238.29,Z 308.124,A -85,B 0,C 180,E1 -19846.647,E2 -19846.647} C_VEL
LIN {X 0,Y 245.403,Z 321.096,A -85,B 0,C 180,E1 -19848.69,E2 -19848.69} C_VEL
LIN {X 0,Y 251.944,Z 334.633,A -85,B 0,C 180,E1 -19850.474,E2 -19850.474} C_VEL
LIN {X 0,Y 258.572,Z 350.298,A -85,B 0,C 180,E1 -19852.214,E2 -19852.214} C_VEL
LIN {X 0,Y 258.51,Z 355.988,A -85,B 0,C 180,E1 -19852.399,E2 -19852.399} C_VEL
LIN {X 0,Y 254.972,Z 430.348,A -85,B 0,C 180,E1 -19854.399,E2 -19854.399} C_VEL
LIN {X 0,Y 253.46,Z 444.897,A -85,B 0,C 180,E1 -19855.058,E2 -19855.058} C_VEL
LIN {X 0,Y 251.604,Z 457.775,A -85,B 0,C 180,E1 -19855.917,E2 -19855.917} C_VEL
LIN {X 0,Y 249.113,Z 471.025,A -85,B 0,C 180,E1 -19857.107,E2 -19857.107} C_VEL
LIN {X 0,Y 246.286,Z 483.797,A -85,B 0,C 180,E1 -19858.616,E2 -19858.616} C_VEL
LIN {X 0,Y 243.42,Z 495.329,A -85,B 0,C 180,E1 -19860.351,E2 -19860.351} C_VEL
LIN {X 0,Y 240.604,Z 505.085,A -85,B 0,C 180,E1 -19862.138,E2 -19862.138} C_VEL
LIN {X 0,Y 237.758,Z 514.174,A -85,B 0,C 180,E1 -19864.152,E2 -19864.152} C_VEL
LIN {X 0,Y 234.8,Z 523.297,A -85,B 0,C 180,E1 -19866.635,E2 -19866.635} C_VEL
LIN {X 0,Y 232.309,Z 530.899,A -85,B 0,C 180,E1 -19869.178,E2 -19869.178} C_VEL
LIN {X 0,Y 229.977,Z 538.157,A -85,B 0,C 180,E1 -19872.207,E2 -19872.207} C_VEL
LIN {X 0,Y 228.353,Z 543.245,A -85,B 0,C 180,E1 -19874.835,E2 -19874.835} C_VEL
LIN {X 0,Y 226.788,Z 548.493,A -85,B 0,C 180,E1 -19878.38,E2 -19878.38} C_VEL
LIN {X 0,Y 226.124,Z 551.436,A -85,B 0,C 180,E1 -19881.06,E2 -19881.06} C_VEL
LIN {X 0,Y 225.646,Z 554.127,A -85,B 0,C 180,E1 -19884.639,E2 -19884.639} C_VEL
LIN {X 0,Y 225.564,Z 555.457,A -85,B 0,C 180,E1 -19888.215,E2 -19888.215} C_VEL
LIN {X 0,Y 225.633,Z 555.62,A -85,B 0,C 180,E1 -19890,E2 -19890} C_VEL
LIN {X 0,Y 225.54,Z 554.943,A -85,B 0,C 180,E1 -19893.573,E2 -19893.573} C_VEL
LIN {X 0,Y 225.821,Z 552.923,A -85,B 0,C 180,E1 -19897.151,E2 -19897.151} C_VEL
LIN {X 0,Y 226.54,Z 549.512,A -85,B 0,C 180,E1 -19900.727,E2 -19900.727} C_VEL
LIN {X 0,Y 227.829,Z 544.607,A -85,B 0,C 180,E1 -19904.287,E2 -19904.287} C_VEL
LIN {X 0,Y 229.4,Z 539.88,A -85,B 0,C 180,E1 -19906.92,E2 -19906.92} C_VEL
LIN {X 0,Y 231.493,Z 533.024,A -85,B 0,C 180,E1 -19909.971,E2 -19909.971} C_VEL
LIN {X 0,Y 234.322,Z 524.516,A -85,B 0,C 180,E1 -19912.948,E2 -19912.948} C_VEL
LIN {X 0,Y 237.251,Z 515.639,A -85,B 0,C 180,E1 -19915.437,E2 -19915.437} C_VEL
LIN {X 0,Y 240.004,Z 506.839,A -85,B 0,C 180,E1 -19917.464,E2 -19917.464} C_VEL
LIN {X 0,Y 243.425,Z 495.087,A -85,B 0,C 180,E1 -19919.649,E2 -19919.649} C_VEL
LIN {X 0,Y 246.283,Z 483.507,A -85,B 0,C 180,E1 -19921.384,E2 -19921.384} C_VEL
LIN {X 0,Y 249.12,Z 470.659,A -85,B 0,C 180,E1 -19922.892,E2 -19922.892} C_VEL
LIN {X 0,Y 251.613,Z 457.294,A -85,B 0,C 180,E1 -19924.081,E2 -19924.081} C_VEL
LIN {X 0,Y 253.555,Z 443.476,A -85,B 0,C 180,E1 -19924.988,E2 -19924.988} C_VEL
LIN {X 0,Y 254.938,Z 430.383,A -85,B 0,C 180,E1 -19925.555,E2 -19925.555} C_VEL
LIN {X 0,Y 258.614,Z 351.623,A -85,B 0,C 180,E1 -19927.681,E2 -19927.681} C_VEL
LIN {X 0,Y 258.365,Z 349.89,A -85,B 0,C 180,E1 -19927.783,E2 -19927.783} C_VEL
LIN {X 0,Y 251.816,Z 334.381,A -85,B 0,C 180,E1 -19929.503,E2 -19929.503} C_VEL
LIN {X 0,Y 245.452,Z 321.31,A -85,B 0,C 180,E1 -19931.23,E2 -19931.23} C_VEL
LIN {X 0,Y 239.598,Z 310.591,A -85,B 0,C 180,E1 -19932.892,E2 -19932.892} C_VEL
LIN {X 0,Y 233.719,Z 300.778,A -85,B 0,C 180,E1 -19934.655,E2 -19934.655} C_VEL
LIN {X 0,Y 230.846,Z 296.327,A -85,B 0,C 180,E1 -19935.555,E2 -19935.555} C_VEL
LIN {X 0,Y 228.657,Z 292.526,A -85,B 0,C 180,E1 -19936.399,E2 -19936.399} C_VEL
LIN {X 0,Y 227.842,Z 289.779,A -85,B 0,C 180,E1 -19937.984,E2 -19937.984} C_VEL
LIN {X 0,Y 227.841,Z 289.72,A -85,B 0,C 180,E1 -19941.908,E2 -19941.908} C_VEL
LIN {X 0,Y 227.876,Z 289.663,A -85,B 0,C 180,E1 -19946.377,E2 -19946.377} C_VEL
LIN {X 0,Y 227.916,Z 289.719,A -85,B 0,C 180,E1 -19950.437,E2 -19950.437} C_VEL
LIN {X 0,Y 227.926,Z 289.715,A -85,B 0,C 180,E1 -19954.426,E2 -19954.426} C_VEL
LIN {X 0,Y 227.959,Z 289.695,A -85,B 0,C 180,E1 -19958.287,E2 -19958.287} C_VEL
LIN {X 0,Y 228.03,Z 289.684,A -85,B 0,C 180,E1 -19962.826,E2 -19962.826} C_VEL
LIN {X 0,Y 228.088,Z 289.691,A -85,B 0,C 180,E1 -19967.544,E2 -19967.544} C_VEL
LIN {X 0,Y 228.302,Z 289.656,A -85,B 0,C 180,E1 -19971.146,E2 -19971.146} C_VEL
LIN {X 0,Y 228.351,Z 289.665,A -85,B 0,C 180,E1 -19972.929,E2 -19972.929} C_VEL
LIN {X 0,Y 228.55,Z 289.634,A -85,B 0,C 180,E1 -19978.238,E2 -19978.238} C_VEL
LIN {X 0,Y 228.55,Z 289.615,A -85,B 0,C 180,E1 -19981.762,E2 -19981.762} C_VEL
LIN {X 0,Y 228.32,Z 289.658,A -85,B 0,C 180,E1 -19987.073,E2 -19987.073} C_VEL
LIN {X 0,Y 228.142,Z 289.679,A -85,B 0,C 180,E1 -19990.652,E2 -19990.652} C_VEL
LIN {X 0,Y 228.058,Z 289.68,A -85,B 0,C 180,E1 -19994.273,E2 -19994.273} C_VEL
LIN {X 0,Y 228,Z 289.71,A -85,B 0,C 180,E1 -19997.954,E2 -19997.954} C_VEL
LIN {X 0,Y 227.927,Z 289.706,A -85,B 0,C 180,E1 -20002.329,E2 -20002.329} C_VEL
LIN {X 0,Y 227.94,Z 289.698,A -85,B 0,C 180,E1 -20006.603,E2 -20006.603} C_VEL
LIN {X 0,Y 227.906,Z 289.697,A -85,B 0,C 180,E1 -20010.297,E2 -20010.297} C_VEL
LIN {X 0,Y 227.887,Z 289.656,A -85,B 0,C 180,E1 -20013.719,E2 -20013.719} C_VEL
LIN {X 0,Y 227.868,Z 289.725,A -85,B 0,C 180,E1 -20018.087,E2 -20018.087} C_VEL
LIN {X 0,Y 227.852,Z 289.788,A -85,B 0,C 180,E1 -20023.11,E2 -20023.11} C_VEL
LIN {X 0,Y 228.045,Z 290.679,A -85,B 0,C 180,E1 -20023.596,E2 -20023.596} C_VEL
LIN {X 0,Y 229.54,Z 293.492,A -85,B 0,C 180,E1 -20024.165,E2 -20024.165} C_VEL
LIN {X 0,Y 231.19,Z 295.365,A -85,B 0,C 180,E1 -20024.667,E2 -20024.667} C_VEL
LIN {X 0,Y 237.404,Z 304.892,A -85,B 0,C 180,E1 -20026.56,E2 -20026.56} C_VEL
LIN {X 0,Y 244.635,Z 317.591,A -85,B 0,C 180,E1 -20028.637,E2 -20028.637} C_VEL
LIN {X 0,Y 251.052,Z 330.246,A -85,B 0,C 180,E1 -20030.38,E2 -20030.38} C_VEL
LIN {X 0,Y 258.26,Z 346.749,A -85,B 0,C 180,E1 -20032.267,E2 -20032.267} C_VEL
LIN {X 0,Y 258.77,Z 348.559,A -85,B 0,C 180,E1 -20032.417,E2 -20032.417} C_VEL
LIN {X 0,Y 254.968,Z 426.634,A -85,B 0,C 180,E1 -20034.503,E2 -20034.503} C_VEL
LIN {X 0,Y 253.473,Z 441.309,A -85,B 0,C 180,E1 -20035.181,E2 -20035.181} C_VEL
LIN {X 0,Y 251.47,Z 455.22,A -85,B 0,C 180,E1 -20036.138,E2 -20036.138} C_VEL
LIN {X 0,Y 249.105,Z 468.166,A -85,B 0,C 180,E1 -20037.346,E2 -20037.346} C_VEL
LIN {X 0,Y 246.409,Z 480.857,A -85,B 0,C 180,E1 -20038.896,E2 -20038.896} C_VEL
LIN {X 0,Y 243.569,Z 492.153,A -85,B 0,C 180,E1 -20040.626,E2 -20040.626} C_VEL
LIN {X 0,Y 240.488,Z 502.655,A -85,B 0,C 180,E1 -20042.596,E2 -20042.596} C_VEL
LIN {X 0,Y 237.256,Z 513.084,A -85,B 0,C 180,E1 -20045.032,E2 -20045.032} C_VEL
LIN {X 0,Y 234.356,Z 521.685,A -85,B 0,C 180,E1 -20047.521,E2 -20047.521} C_VEL
LIN {X 0,Y 231.672,Z 529.927,A -85,B 0,C 180,E1 -20050.507,E2 -20050.507} C_VEL
LIN {X 0,Y 229.843,Z 535.671,A -85,B 0,C 180,E1 -20053.113,E2 -20053.113} C_VEL
LIN {X 0,Y 228.159,Z 540.393,A -85,B 0,C 180,E1 -20055.734,E2 -20055.734} C_VEL
LIN {X 0,Y 226.783,Z 545.283,A -85,B 0,C 180,E1 -20059.284,E2 -20059.284} C_VEL
LIN {X 0,Y 226,Z 548.683,A -85,B 0,C 180,E1 -20062.855,E2 -20062.855} C_VEL
LIN {X 0,Y 225.629,Z 550.7,A -85,B 0,C 180,E1 -20066.428,E2 -20066.428} C_VEL
LIN {X 0,Y 225.637,Z 551.387,A -85,B 0,C 180,E1 -20070,E2 -20070} C_VEL
LIN {X 0,Y 225.629,Z 550.755,A -85,B 0,C 180,E1 -20073.571,E2 -20073.571} C_VEL
LIN {X 0,Y 225.997,Z 548.787,A -85,B 0,C 180,E1 -20077.145,E2 -20077.145} C_VEL
LIN {X 0,Y 226.763,Z 545.437,A -85,B 0,C 180,E1 -20080.717,E2 -20080.717} C_VEL
LIN {X 0,Y 228.135,Z 540.606,A -85,B 0,C 180,E1 -20084.267,E2 -20084.267} C_VEL
LIN {X 0,Y 230.392,Z 534.135,A -85,B 0,C 180,E1 -20087.76,E2 -20087.76} C_VEL
LIN {X 0,Y 232.413,Z 527.63,A -85,B 0,C 180,E1 -20090.521,E2 -20090.521} C_VEL
LIN {X 0,Y 235.196,Z 519.381,A -85,B 0,C 180,E1 -20093.323,E2 -20093.323} C_VEL
LIN {X 0,Y 238.181,Z 510.312,A -85,B 0,C 180,E1 -20095.799,E2 -20095.799} C_VEL
LIN {X 0,Y 241.583,Z 499.326,A -85,B 0,C 180,E1 -20098.211,E2 -20098.211} C_VEL
LIN {X 0,Y 244.917,Z 487.48,A -85,B 0,C 180,E1 -20100.26,E2 -20100.26} C_VEL
LIN {X 0,Y 247.54,Z 476.186,A -85,B 0,C 180,E1 -20101.851,E2 -20101.851} C_VEL
LIN {X 0,Y 250.135,Z 463.761,A -85,B 0,C 180,E1 -20103.221,E2 -20103.221} C_VEL
LIN {X 0,Y 252.342,Z 450.665,A -85,B 0,C 180,E1 -20104.331,E2 -20104.331} C_VEL
LIN {X 0,Y 254.097,Z 437.415,A -85,B 0,C 180,E1 -20105.144,E2 -20105.144} C_VEL
LIN {X 0,Y 255.297,Z 423.031,A -85,B 0,C 180,E1 -20105.737,E2 -20105.737} C_VEL
LIN {X 0,Y 258.477,Z 356.396,A -85,B 0,C 180,E1 -20107.505,E2 -20107.505} C_VEL
LIN {X 0,Y 258.769,Z 347.885,A -85,B 0,C 180,E1 -20107.748,E2 -20107.748} C_VEL
LIN {X 0,Y 252.18,Z 332.6,A -85,B 0,C 180,E1 -20109.469,E2 -20109.469} C_VEL
LIN {X 0,Y 244.912,Z 318.011,A -85,B 0,C 180,E1 -20111.442,E2 -20111.442} C_VEL
LIN {X 0,Y 238.106,Z 306.156,A -85,B 0,C 180,E1 -20113.388,E2 -20113.388} C_VEL
LIN {X 0,Y 233.413,Z 298.6,A -85,B 0,C 180,E1 -20114.809,E2 -20114.809} C_VEL
LIN {X 0,Y 231.215,Z 295.399,A -85,B 0,C 180,E1 -20115.492,E2 -20115.492} C_VEL
LIN {X 0,Y 230.038,Z 294.019,A -85,B 0,C 180,E1 -20115.852,E2 -20115.852} C_VEL
LIN {X 0,Y 228.368,Z 291.589,A -85,B 0,C 180,E1 -20116.405,E2 -20116.405} C_VEL
LIN {X 0,Y 227.925,Z 290.178,A -85,B 0,C 180,E1 -20116.756,E2 -20116.756} C_VEL
LIN {X 0,Y 227.82,Z 289.744,A -85,B 0,C 180,E1 -20117.259,E2 -20117.259} C_VEL
LIN {X 0,Y 227.868,Z 289.725,A -85,B 0,C 180,E1 -20121.913,E2 -20121.913} C_VEL
LIN {X 0,Y 227.887,Z 289.66,A -85,B 0,C 180,E1 -20126.373,E2 -20126.373} C_VEL
LIN {X 0,Y 227.916,Z 289.714,A -85,B 0,C 180,E1 -20130.437,E2 -20130.437} C_VEL
LIN {X 0,Y 227.925,Z 289.702,A -85,B 0,C 180,E1 -20134.425,E2 -20134.425} C_VEL
LIN {X 0,Y 227.958,Z 289.697,A -85,B 0,C 180,E1 -20138.286,E2 -20138.286} C_VEL
LIN {X 0,Y 228.03,Z 289.702,A -85,B 0,C 180,E1 -20142.826,E2 -20142.826} C_VEL
LIN {X 0,Y 228.067,Z 289.699,A -85,B 0,C 180,E1 -20147.543,E2 -20147.543} C_VEL
LIN {X 0,Y 228.262,Z 289.651,A -85,B 0,C 180,E1 -20151.144,E2 -20151.144} C_VEL
LIN {X 0,Y 228.319,Z 289.657,A -85,B 0,C 180,E1 -20152.927,E2 -20152.927} C_VEL
LIN {X 0,Y 228.55,Z 289.615,A -85,B 0,C 180,E1 -20158.238,E2 -20158.238} C_VEL
LIN {X 0,Y 228.549,Z 289.634,A -85,B 0,C 180,E1 -20161.762,E2 -20161.762} C_VEL
LIN {X 0,Y 228.35,Z 289.666,A -85,B 0,C 180,E1 -20167.071,E2 -20167.071} C_VEL
LIN {X 0,Y 228.158,Z 289.665,A -85,B 0,C 180,E1 -20170.65,E2 -20170.65} C_VEL
LIN {X 0,Y 228.055,Z 289.698,A -85,B 0,C 180,E1 -20174.273,E2 -20174.273} C_VEL
LIN {X 0,Y 227.994,Z 289.697,A -85,B 0,C 180,E1 -20177.993,E2 -20177.993} C_VEL
LIN {X 0,Y 227.223,Z 289.807,A -85,B 0,C 180,E1 -20179.467,E2 -20179.467} C_VEL
LIN {X 0,Y 224.301,Z 290.16,A -85,B 0,C 180,E1 -20181.871,E2 -20181.871} C_VEL
LIN {X 0,Y 221.901,Z 290.46,A -85,B 0,C 180,E1 -20183.834,E2 -20183.834} C_VEL
LIN {X 0,Y 220.916,Z 290.59,A -85,B 0,C 180,E1 -20185.358,E2 -20185.358} C_VEL
LIN {X 0,Y 220.855,Z 290.585,A -85,B 0,C 180,E1 -20185.874,E2 -20185.874} C_VEL
LIN {X 0,Y 220.86,Z 290.588,A -85,B 0,C 180,E1 -20190.779,E2 -20190.779} C_VEL
LIN {X 0,Y 220.797,Z 290.542,A -85,B 0,C 180,E1 -20194.956,E2 -20194.956} C_VEL
LIN {X 0,Y 220.804,Z 290.597,A -85,B 0,C 180,E1 -20199.537,E2 -20199.537} C_VEL
LIN {X 0,Y 220.804,Z 290.759,A -85,B 0,C 180,E1 -20200.505,E2 -20200.505} C_VEL
LIN {X 0,Y 221.468,Z 292.827,A -85,B 0,C 180,E1 -20201.61,E2 -20201.61} C_VEL
LIN {X 0,Y 224.293,Z 297.193,A -85,B 0,C 180,E1 -20202.672,E2 -20202.672} C_VEL
LIN {X 0,Y 229.891,Z 305.924,A -85,B 0,C 180,E1 -20204.545,E2 -20204.545} C_VEL
LIN {X 0,Y 236.51,Z 317.103,A -85,B 0,C 180,E1 -20206.608,E2 -20206.608} C_VEL
LIN {X 0,Y 243.884,Z 331.483,A -85,B 0,C 180,E1 -20208.775,E2 -20208.775} C_VEL
LIN {X 0,Y 251.626,Z 349.141,A -85,B 0,C 180,E1 -20210.938,E2 -20210.938} C_VEL
LIN {X 0,Y 253.05,Z 352.696,A -85,B 0,C 180,E1 -20211.326,E2 -20211.326} C_VEL
LIN {X 0,Y 249.306,Z 429.589,A -85,B 0,C 180,E1 -20213.427,E2 -20213.427} C_VEL
LIN {X 0,Y 247.784,Z 444.077,A -85,B 0,C 180,E1 -20214.073,E2 -20214.073} C_VEL
LIN {X 0,Y 245.761,Z 457.715,A -85,B 0,C 180,E1 -20214.991,E2 -20214.991} C_VEL
LIN {X 0,Y 243.193,Z 470.964,A -85,B 0,C 180,E1 -20216.2,E2 -20216.2} C_VEL
LIN {X 0,Y 240.238,Z 483.735,A -85,B 0,C 180,E1 -20217.732,E2 -20217.732} C_VEL
LIN {X 0,Y 237.424,Z 494.778,A -85,B 0,C 180,E1 -20219.422,E2 -20219.422} C_VEL
LIN {X 0,Y 234.327,Z 505.022,A -85,B 0,C 180,E1 -20221.323,E2 -20221.323} C_VEL
LIN {X 0,Y 230.827,Z 515.739,A -85,B 0,C 180,E1 -20223.802,E2 -20223.802} C_VEL
LIN {X 0,Y 227.784,Z 524.588,A -85,B 0,C 180,E1 -20226.354,E2 -20226.354} C_VEL
LIN {X 0,Y 225.259,Z 531.952,A -85,B 0,C 180,E1 -20228.974,E2 -20228.974} C_VEL
LIN {X 0,Y 223.198,Z 538.092,A -85,B 0,C 180,E1 -20231.647,E2 -20231.647} C_VEL
LIN {X 0,Y 221.461,Z 543.179,A -85,B 0,C 180,E1 -20234.351,E2 -20234.351} C_VEL
LIN {X 0,Y 219.789,Z 548.427,A -85,B 0,C 180,E1 -20238.004,E2 -20238.004} C_VEL
LIN {X 0,Y 219.074,Z 551.37,A -85,B 0,C 180,E1 -20240.77,E2 -20240.77} C_VEL
LIN {X 0,Y 218.568,Z 554.061,A -85,B 0,C 180,E1 -20244.465,E2 -20244.465} C_VEL
LIN {X 0,Y 218.466,Z 555.39,A -85,B 0,C 180,E1 -20248.157,E2 -20248.157} C_VEL
LIN {X 0,Y 218.532,Z 555.554,A -85,B 0,C 180,E1 -20250,E2 -20250} C_VEL
LIN {X 0,Y 218.449,Z 554.876,A -85,B 0,C 180,E1 -20253.689,E2 -20253.689} C_VEL
LIN {X 0,Y 218.758,Z 552.856,A -85,B 0,C 180,E1 -20257.383,E2 -20257.383} C_VEL
LIN {X 0,Y 219.545,Z 549.445,A -85,B 0,C 180,E1 -20261.073,E2 -20261.073} C_VEL
LIN {X 0,Y 220.938,Z 544.539,A -85,B 0,C 180,E1 -20264.742,E2 -20264.742} C_VEL
LIN {X 0,Y 222.554,Z 539.811,A -85,B 0,C 180,E1 -20267.457,E2 -20267.457} C_VEL
LIN {X 0,Y 224.786,Z 532.955,A -85,B 0,C 180,E1 -20270.593,E2 -20270.593} C_VEL
LIN {X 0,Y 227.775,Z 524.448,A -85,B 0,C 180,E1 -20273.648,E2 -20273.648} C_VEL
LIN {X 0,Y 230.802,Z 515.57,A -85,B 0,C 180,E1 -20276.201,E2 -20276.201} C_VEL
LIN {X 0,Y 233.719,Z 506.77,A -85,B 0,C 180,E1 -20278.268,E2 -20278.268} C_VEL
LIN {X 0,Y 236.891,Z 496.28,A -85,B 0,C 180,E1 -20280.288,E2 -20280.288} C_VEL
LIN {X 0,Y 239.872,Z 484.863,A -85,B 0,C 180,E1 -20282.075,E2 -20282.075} C_VEL
LIN {X 0,Y 242.795,Z 472.354,A -85,B 0,C 180,E1 -20283.613,E2 -20283.613} C_VEL
LIN {X 0,Y 245.347,Z 459.481,A -85,B 0,C 180,E1 -20284.827,E2 -20284.827} C_VEL
LIN {X 0,Y 247.559,Z 444.938,A -85,B 0,C 180,E1 -20285.839,E2 -20285.839} C_VEL
LIN {X 0,Y 248.982,Z 432.097,A -85,B 0,C 180,E1 -20286.442,E2 -20286.442} C_VEL
LIN {X 0,Y 250.404,Z 405.419,A -85,B 0,C 180,E1 -20287.222,E2 -20287.222} C_VEL
LIN {X 0,Y 252.93,Z 352.585,A -85,B 0,C 180,E1 -20288.645,E2 -20288.645} C_VEL
LIN {X 0,Y 246.482,Z 337.228,A -85,B 0,C 180,E1 -20290.423,E2 -20290.423} C_VEL
LIN {X 0,Y 239.969,Z 323.723,A -85,B 0,C 180,E1 -20292.289,E2 -20292.289} C_VEL
LIN {X 0,Y 233.258,Z 311.61,A -85,B 0,C 180,E1 -20294.309,E2 -20294.309} C_VEL
LIN {X 0,Y 227.682,Z 302.383,A -85,B 0,C 180,E1 -20296.1,E2 -20296.1} C_VEL
LIN {X 0,Y 223.551,Z 296.298,A -85,B 0,C 180,E1 -20297.49,E2 -20297.49} C_VEL
LIN {X 0,Y 221.261,Z 292.393,A -85,B 0,C 180,E1 -20298.463,E2 -20298.463} C_VEL
LIN {X 0,Y 220.804,Z 290.688,A -85,B 0,C 180,E1 -20299.496,E2 -20299.496} C_VEL
LIN {X 0,Y 220.822,Z 290.568,A -85,B 0,C 180,E1 -20302.793,E2 -20302.793} C_VEL
LIN {X 0,Y 220.815,Z 290.551,A -85,B 0,C 180,E1 -20307.244,E2 -20307.244} C_VEL
LIN {X 0,Y 220.833,Z 290.587,A -85,B 0,C 180,E1 -20311.486,E2 -20311.486} C_VEL
LIN {X 0,Y 220.864,Z 290.596,A -85,B 0,C 180,E1 -20315.565,E2 -20315.565} C_VEL
LIN {X 0,Y 220.889,Z 290.586,A -85,B 0,C 180,E1 -20319.514,E2 -20319.514} C_VEL
LIN {X 0,Y 221.011,Z 290.556,A -85,B 0,C 180,E1 -20323.37,E2 -20323.37} C_VEL
LIN {X 0,Y 221.108,Z 290.544,A -85,B 0,C 180,E1 -20329.006,E2 -20329.006} C_VEL
LIN {X 0,Y 221.302,Z 290.543,A -85,B 0,C 180,E1 -20332.702,E2 -20332.702} C_VEL
LIN {X 0,Y 221.508,Z 290.51,A -85,B 0,C 180,E1 -20338.182,E2 -20338.182} C_VEL
LIN {X 0,Y 221.508,Z 290.491,A -85,B 0,C 180,E1 -20341.818,E2 -20341.818} C_VEL
LIN {X 0,Y 221.255,Z 290.533,A -85,B 0,C 180,E1 -20347.3,E2 -20347.3} C_VEL
LIN {X 0,Y 221.078,Z 290.564,A -85,B 0,C 180,E1 -20350.996,E2 -20350.996} C_VEL
LIN {X 0,Y 221.013,Z 290.566,A -85,B 0,C 180,E1 -20356.63,E2 -20356.63} C_VEL
LIN {X 0,Y 220.889,Z 290.574,A -85,B 0,C 180,E1 -20360.487,E2 -20360.487} C_VEL
LIN {X 0,Y 220.865,Z 290.592,A -85,B 0,C 180,E1 -20364.436,E2 -20364.436} C_VEL
LIN {X 0,Y 220.835,Z 290.602,A -85,B 0,C 180,E1 -20368.514,E2 -20368.514} C_VEL
LIN {X 0,Y 220.822,Z 290.537,A -85,B 0,C 180,E1 -20372.756,E2 -20372.756} C_VEL
LIN {X 0,Y 220.837,Z 290.594,A -85,B 0,C 180,E1 -20377.289,E2 -20377.289} C_VEL
LIN {X 0,Y 220.785,Z 290.729,A -85,B 0,C 180,E1 -20381.226,E2 -20381.226} C_VEL
LIN {X 0,Y 221.014,Z 291.755,A -85,B 0,C 180,E1 -20381.715,E2 -20381.715} C_VEL
LIN {X 0,Y 222.549,Z 294.42,A -85,B 0,C 180,E1 -20382.317,E2 -20382.317} C_VEL
LIN {X 0,Y 224.328,Z 296.35,A -85,B 0,C 180,E1 -20382.904,E2 -20382.904} C_VEL
LIN {X 0,Y 226.636,Z 299.727,A -85,B 0,C 180,E1 -20383.683,E2 -20383.683} C_VEL
LIN {X 0,Y 231.301,Z 306.564,A -85,B 0,C 180,E1 -20385.178,E2 -20385.178} C_VEL
LIN {X 0,Y 238.02,Z 318.015,A -85,B 0,C 180,E1 -20387.232,E2 -20387.232} C_VEL
LIN {X 0,Y 245,Z 331.522,A -85,B 0,C 180,E1 -20389.243,E2 -20389.243} C_VEL
LIN {X 0,Y 252.445,Z 348.441,A -85,B 0,C 180,E1 -20391.296,E2 -20391.296} C_VEL
LIN {X 0,Y 253.011,Z 349.906,A -85,B 0,C 180,E1 -20391.451,E2 -20391.451} C_VEL
LIN {X 0,Y 249.917,Z 415.222,A -85,B 0,C 180,E1 -20393.216,E2 -20393.216} C_VEL
LIN {X 0,Y 248.97,Z 430.271,A -85,B 0,C 180,E1 -20393.708,E2 -20393.708} C_VEL
LIN {X 0,Y 247.29,Z 444.431,A -85,B 0,C 180,E1 -20394.429,E2 -20394.429} C_VEL
LIN {X 0,Y 245.041,Z 458.673,A -85,B 0,C 180,E1 -20395.498,E2 -20395.498} C_VEL
LIN {X 0,Y 242.447,Z 471.709,A -85,B 0,C 180,E1 -20396.83,E2 -20396.83} C_VEL
LIN {X 0,Y 239.793,Z 483.325,A -85,B 0,C 180,E1 -20398.361,E2 -20398.361} C_VEL
LIN {X 0,Y 236.42,Z 495.584,A -85,B 0,C 180,E1 -20400.383,E2 -20400.383} C_VEL
LIN {X 0,Y 232.992,Z 506.42,A -85,B 0,C 180,E1 -20402.613,E2 -20402.613} C_VEL
LIN {X 0,Y 229.799,Z 516.172,A -85,B 0,C 180,E1 -20405.133,E2 -20405.133} C_VEL
LIN {X 0,Y 226.877,Z 524.263,A -85,B 0,C 180,E1 -20407.7,E2 -20407.7} C_VEL
LIN {X 0,Y 224.258,Z 532.006,A -85,B 0,C 180,E1 -20410.789,E2 -20410.789} C_VEL
LIN {X 0,Y 222.397,Z 537.414,A -85,B 0,C 180,E1 -20413.477,E2 -20413.477} C_VEL
LIN {X 0,Y 220.835,Z 541.861,A -85,B 0,C 180,E1 -20416.191,E2 -20416.191} C_VEL
LIN {X 0,Y 219.772,Z 545.35,A -85,B 0,C 180,E1 -20418.938,E2 -20418.938} C_VEL
LIN {X 0,Y 218.943,Z 548.751,A -85,B 0,C 180,E1 -20422.623,E2 -20422.623} C_VEL
LIN {X 0,Y 218.534,Z 550.767,A -85,B 0,C 180,E1 -20426.312,E2 -20426.312} C_VEL
LIN {X 0,Y 218.537,Z 551.454,A -85,B 0,C 180,E1 -20430,E2 -20430} C_VEL
LIN {X 0,Y 218.535,Z 550.822,A -85,B 0,C 180,E1 -20433.688,E2 -20433.688} C_VEL
LIN {X 0,Y 218.941,Z 548.853,A -85,B 0,C 180,E1 -20437.377,E2 -20437.377} C_VEL
LIN {X 0,Y 219.751,Z 545.503,A -85,B 0,C 180,E1 -20441.063,E2 -20441.063} C_VEL
LIN {X 0,Y 221.226,Z 540.671,A -85,B 0,C 180,E1 -20444.723,E2 -20444.723} C_VEL
LIN {X 0,Y 222.971,Z 536.005,A -85,B 0,C 180,E1 -20447.423,E2 -20447.423} C_VEL
LIN {X 0,Y 225.269,Z 529.059,A -85,B 0,C 180,E1 -20450.617,E2 -20450.617} C_VEL
LIN {X 0,Y 228.193,Z 520.797,A -85,B 0,C 180,E1 -20453.601,E2 -20453.601} C_VEL
LIN {X 0,Y 231.23,Z 512.001,A -85,B 0,C 180,E1 -20456.149,E2 -20456.149} C_VEL
LIN {X 0,Y 234.705,Z 501.341,A -85,B 0,C 180,E1 -20458.626,E2 -20458.626} C_VEL
LIN {X 0,Y 238.172,Z 489.878,A -85,B 0,C 180,E1 -20460.74,E2 -20460.74} C_VEL
LIN {X 0,Y 241.298,Z 477.333,A -85,B 0,C 180,E1 -20462.602,E2 -20462.602} C_VEL
LIN {X 0,Y 243.854,Z 465.726,A -85,B 0,C 180,E1 -20463.944,E2 -20463.944} C_VEL
LIN {X 0,Y 246.129,Z 453.216,A -85,B 0,C 180,E1 -20465.074,E2 -20465.074} C_VEL
LIN {X 0,Y 248.144,Z 439.29,A -85,B 0,C 180,E1 -20465.992,E2 -20465.992} C_VEL
LIN {X 0,Y 249.476,Z 424.683,A -85,B 0,C 180,E1 -20466.637,E2 -20466.637} C_VEL
LIN {X 0,Y 252.805,Z 358.359,A -85,B 0,C 180,E1 -20468.43,E2 -20468.43} C_VEL
LIN {X 0,Y 253.077,Z 349.919,A -85,B 0,C 180,E1 -20468.682,E2 -20468.682} C_VEL
LIN {X 0,Y 247.087,Z 335.968,A -85,B 0,C 180,E1 -20470.324,E2 -20470.324} C_VEL
LIN {X 0,Y 240.189,Z 321.942,A -85,B 0,C 180,E1 -20472.29,E2 -20472.29} C_VEL
LIN {X 0,Y 232.781,Z 308.861,A -85,B 0,C 180,E1 -20474.527,E2 -20474.527} C_VEL
LIN {X 0,Y 229.326,Z 303.53,A -85,B 0,C 180,E1 -20475.617,E2 -20475.617} C_VEL
LIN {X 0,Y 226.625,Z 299.694,A -85,B 0,C 180,E1 -20476.493,E2 -20476.493} C_VEL
LIN {X 0,Y 224.374,Z 296.451,A -85,B 0,C 180,E1 -20477.253,E2 -20477.253} C_VEL
LIN {X 0,Y 223.678,Z 295.465,A -85,B 0,C 180,E1 -20477.492,E2 -20477.492} C_VEL
LIN {X 0,Y 221.607,Z 293.163,A -85,B 0,C 180,E1 -20478.19,E2 -20478.19} C_VEL
LIN {X 0,Y 220.843,Z 291.111,A -85,B 0,C 180,E1 -20478.667,E2 -20478.667} C_VEL
LIN {X 0,Y 220.788,Z 290.647,A -85,B 0,C 180,E1 -20479.014,E2 -20479.014} C_VEL
LIN {X 0,Y 220.83,Z 290.602,A -85,B 0,C 180,E1 -20482.794,E2 -20482.794} C_VEL
LIN {X 0,Y 220.821,Z 290.54,A -85,B 0,C 180,E1 -20487.244,E2 -20487.244} C_VEL
LIN {X 0,Y 220.834,Z 290.605,A -85,B 0,C 180,E1 -20491.486,E2 -20491.486} C_VEL
LIN {X 0,Y 220.864,Z 290.591,A -85,B 0,C 180,E1 -20495.564,E2 -20495.564} C_VEL
LIN {X 0,Y 220.888,Z 290.574,A -85,B 0,C 180,E1 -20499.513,E2 -20499.513} C_VEL
LIN {X 0,Y 221.012,Z 290.568,A -85,B 0,C 180,E1 -20503.37,E2 -20503.37} C_VEL
LIN {X 0,Y 221.077,Z 290.566,A -85,B 0,C 180,E1 -20509.004,E2 -20509.004} C_VEL
LIN {X 0,Y 221.254,Z 290.533,A -85,B 0,C 180,E1 -20512.7,E2 -20512.7} C_VEL
LIN {X 0,Y 221.507,Z 290.491,A -85,B 0,C 180,E1 -20518.182,E2 -20518.182} C_VEL
LIN {X 0,Y 221.507,Z 290.51,A -85,B 0,C 180,E1 -20521.818,E2 -20521.818} C_VEL
LIN {X 0,Y 221.301,Z 290.543,A -85,B 0,C 180,E1 -20527.298,E2 -20527.298} C_VEL
LIN {X 0,Y 221.107,Z 290.544,A -85,B 0,C 180,E1 -20530.994,E2 -20530.994} C_VEL
LIN {X 0,Y 221.01,Z 290.557,A -85,B 0,C 180,E1 -20536.63,E2 -20536.63} C_VEL
LIN {X 0,Y 220.888,Z 290.586,A -85,B 0,C 180,E1 -20540.486,E2 -20540.486} C_VEL
LIN {X 0,Y 220.864,Z 290.597,A -85,B 0,C 180,E1 -20544.435,E2 -20544.435} C_VEL
LIN {X 0,Y 220.855,Z 290.585,A -85,B 0,C 180,E1 -20545.874,E2 -20545.874} C_VEL
LIN {X 0,Y 220.575,Z 290.622,A -85,B 0,C 180,E1 -20546.892,E2 -20546.892} C_VEL
LIN {X 0,Y 219.249,Z 290.8,A -85,B 0,C 180,E1 -20548.396,E2 -20548.396} C_VEL
LIN {X 0,Y 214.895,Z 291.307,A -85,B 0,C 180,E1 -20551.909,E2 -20551.909} C_VEL
LIN {X 0,Y 213.837,Z 291.411,A -85,B 0,C 180,E1 -20553.486,E2 -20553.486} C_VEL
LIN {X 0,Y 213.753,Z 291.418,A -85,B 0,C 180,E1 -20554.021,E2 -20554.021} C_VEL
LIN {X 0,Y 213.756,Z 291.613,A -85,B 0,C 180,E1 -20558.735,E2 -20558.735} C_VEL
LIN {X 0,Y 214.075,Z 292.883,A -85,B 0,C 180,E1 -20559.347,E2 -20559.347} C_VEL
LIN {X 0,Y 215.767,Z 295.613,A -85,B 0,C 180,E1 -20560.08,E2 -20560.08} C_VEL
LIN {X 0,Y 218.49,Z 299.318,A -85,B 0,C 180,E1 -20561.102,E2 -20561.102} C_VEL
LIN {X 0,Y 224.88,Z 309.069,A -85,B 0,C 180,E1 -20563.377,E2 -20563.377} C_VEL
LIN {X 0,Y 232.123,Z 321.537,A -85,B 0,C 180,E1 -20565.764,E2 -20565.764} C_VEL
LIN {X 0,Y 239.102,Z 335.329,A -85,B 0,C 180,E1 -20567.917,E2 -20567.917} C_VEL
LIN {X 0,Y 246.518,Z 352.424,A -85,B 0,C 180,E1 -20570.092,E2 -20570.092} C_VEL
LIN {X 0,Y 247.404,Z 354.72,A -85,B 0,C 180,E1 -20570.348,E2 -20570.348} C_VEL
LIN {X 0,Y 243.624,Z 429.861,A -85,B 0,C 180,E1 -20572.444,E2 -20572.444} C_VEL
LIN {X 0,Y 242.087,Z 444.02,A -85,B 0,C 180,E1 -20573.09,E2 -20573.09} C_VEL
LIN {X 0,Y 240.18,Z 456.522,A -85,B 0,C 180,E1 -20573.923,E2 -20573.923} C_VEL
LIN {X 0,Y 237.714,Z 469.135,A -85,B 0,C 180,E1 -20575.054,E2 -20575.054} C_VEL
LIN {X 0,Y 234.628,Z 482.246,A -85,B 0,C 180,E1 -20576.607,E2 -20576.607} C_VEL
LIN {X 0,Y 231.566,Z 493.736,A -85,B 0,C 180,E1 -20578.349,E2 -20578.349} C_VEL
LIN {X 0,Y 228.106,Z 504.958,A -85,B 0,C 180,E1 -20580.465,E2 -20580.465} C_VEL
LIN {X 0,Y 224.451,Z 515.674,A -85,B 0,C 180,E1 -20582.999,E2 -20582.999} C_VEL
LIN {X 0,Y 221.271,Z 524.523,A -85,B 0,C 180,E1 -20585.613,E2 -20585.613} C_VEL
LIN {X 0,Y 218.203,Z 533.004,A -85,B 0,C 180,E1 -20588.756,E2 -20588.756} C_VEL
LIN {X 0,Y 215.759,Z 539.839,A -85,B 0,C 180,E1 -20591.975,E2 -20591.975} C_VEL
LIN {X 0,Y 214.06,Z 544.548,A -85,B 0,C 180,E1 -20594.773,E2 -20594.773} C_VEL
LIN {X 0,Y 212.521,Z 549.428,A -85,B 0,C 180,E1 -20598.556,E2 -20598.556} C_VEL
LIN {X 0,Y 211.684,Z 552.822,A -85,B 0,C 180,E1 -20602.369,E2 -20602.369} C_VEL
LIN {X 0,Y 211.349,Z 554.827,A -85,B 0,C 180,E1 -20606.187,E2 -20606.187} C_VEL
LIN {X 0,Y 211.433,Z 555.487,A -85,B 0,C 180,E1 -20610,E2 -20610} C_VEL
LIN {X 0,Y 211.349,Z 554.809,A -85,B 0,C 180,E1 -20613.813,E2 -20613.813} C_VEL
LIN {X 0,Y 211.685,Z 552.789,A -85,B 0,C 180,E1 -20617.631,E2 -20617.631} C_VEL
LIN {X 0,Y 212.525,Z 549.377,A -85,B 0,C 180,E1 -20621.444,E2 -20621.444} C_VEL
LIN {X 0,Y 214.06,Z 544.472,A -85,B 0,C 180,E1 -20625.227,E2 -20625.227} C_VEL
LIN {X 0,Y 215.733,Z 539.743,A -85,B 0,C 180,E1 -20628.028,E2 -20628.028} C_VEL
LIN {X 0,Y 218.108,Z 532.887,A -85,B 0,C 180,E1 -20631.254,E2 -20631.254} C_VEL
LIN {X 0,Y 221.258,Z 524.379,A -85,B 0,C 180,E1 -20634.389,E2 -20634.389} C_VEL
LIN {X 0,Y 224.41,Z 515.5,A -85,B 0,C 180,E1 -20637.007,E2 -20637.007} C_VEL
LIN {X 0,Y 228.117,Z 504.747,A -85,B 0,C 180,E1 -20639.533,E2 -20639.533} C_VEL
LIN {X 0,Y 231.594,Z 493.413,A -85,B 0,C 180,E1 -20641.662,E2 -20641.662} C_VEL
LIN {X 0,Y 234.61,Z 481.939,A -85,B 0,C 180,E1 -20643.397,E2 -20643.397} C_VEL
LIN {X 0,Y 237.728,Z 468.728,A -85,B 0,C 180,E1 -20644.944,E2 -20644.944} C_VEL
LIN {X 0,Y 240.186,Z 455.981,A -85,B 0,C 180,E1 -20646.076,E2 -20646.076} C_VEL
LIN {X 0,Y 242.228,Z 441.532,A -85,B 0,C 180,E1 -20647.015,E2 -20647.015} C_VEL
LIN {X 0,Y 243.726,Z 426.775,A -85,B 0,C 180,E1 -20647.615,E2 -20647.615} C_VEL
LIN {X 0,Y 247.3,Z 355.776,A -85,B 0,C 180,E1 -20649.575,E2 -20649.575} C_VEL
LIN {X 0,Y 247.063,Z 354.084,A -85,B 0,C 180,E1 -20649.683,E2 -20649.683} C_VEL
LIN {X 0,Y 241.487,Z 340.656,A -85,B 0,C 180,E1 -20651.304,E2 -20651.304} C_VEL
LIN {X 0,Y 234.667,Z 326.554,A -85,B 0,C 180,E1 -20653.357,E2 -20653.357} C_VEL
LIN {X 0,Y 228.863,Z 315.95,A -85,B 0,C 180,E1 -20655.201,E2 -20655.201} C_VEL
LIN {X 0,Y 223.402,Z 306.897,A -85,B 0,C 180,E1 -20657.041,E2 -20657.041} C_VEL
LIN {X 0,Y 219.729,Z 301.356,A -85,B 0,C 180,E1 -20658.342,E2 -20658.342} C_VEL
LIN {X 0,Y 216.561,Z 296.549,A -85,B 0,C 180,E1 -20659.53,E2 -20659.53} C_VEL
LIN {X 0,Y 214.341,Z 293.544,A -85,B 0,C 180,E1 -20660.407,E2 -20660.407} C_VEL
LIN {X 0,Y 213.884,Z 292.257,A -85,B 0,C 180,E1 -20660.763,E2 -20660.763} C_VEL
LIN {X 0,Y 213.744,Z 291.561,A -85,B 0,C 180,E1 -20661.338,E2 -20661.338} C_VEL
LIN {X 0,Y 213.754,Z 291.418,A -85,B 0,C 180,E1 -20666.017,E2 -20666.017} C_VEL
LIN {X 0,Y 213.778,Z 291.479,A -85,B 0,C 180,E1 -20670.454,E2 -20670.454} C_VEL
LIN {X 0,Y 213.799,Z 291.477,A -85,B 0,C 180,E1 -20674.702,E2 -20674.702} C_VEL
LIN {X 0,Y 213.809,Z 291.459,A -85,B 0,C 180,E1 -20678.803,E2 -20678.803} C_VEL
LIN {X 0,Y 213.939,Z 291.439,A -85,B 0,C 180,E1 -20682.803,E2 -20682.803} C_VEL
LIN {X 0,Y 213.974,Z 291.457,A -85,B 0,C 180,E1 -20686.708,E2 -20686.708} C_VEL
LIN {X 0,Y 214.164,Z 291.41,A -85,B 0,C 180,E1 -20690.556,E2 -20690.556} C_VEL
LIN {X 0,Y 214.236,Z 291.423,A -85,B 0,C 180,E1 -20692.46,E2 -20692.46} C_VEL
LIN {X 0,Y 214.441,Z 291.389,A -85,B 0,C 180,E1 -20698.122,E2 -20698.122} C_VEL
LIN {X 0,Y 214.546,Z 291.381,A -85,B 0,C 180,E1 -20700,E2 -20700} C_VEL
LIN {X 0,Y 214.441,Z 291.371,A -85,B 0,C 180,E1 -20701.878,E2 -20701.878} C_VEL
LIN {X 0,Y 214.194,Z 291.409,A -85,B 0,C 180,E1 -20707.542,E2 -20707.542} C_VEL
LIN {X 0,Y 214.004,Z 291.449,A -85,B 0,C 180,E1 -20711.364,E2 -20711.364} C_VEL
LIN {X 0,Y 213.928,Z 291.437,A -85,B 0,C 180,E1 -20715.238,E2 -20715.238} C_VEL
LIN {X 0,Y 213.836,Z 291.463,A -85,B 0,C 180,E1 -20719.188,E2 -20719.188} C_VEL
LIN {X 0,Y 213.845,Z 291.471,A -85,B 0,C 180,E1 -20723.228,E2 -20723.228} C_VEL
LIN {X 0,Y 213.827,Z 291.46,A -85,B 0,C 180,E1 -20727.45,E2 -20727.45} C_VEL
LIN {X 0,Y 213.777,Z 291.423,A -85,B 0,C 180,E1 -20731.736,E2 -20731.736} C_VEL
LIN {X 0,Y 213.751,Z 291.447,A -85,B 0,C 180,E1 -20736.287,E2 -20736.287} C_VEL
LIN {X 0,Y 213.786,Z 291.726,A -85,B 0,C 180,E1 -20739.221,E2 -20739.221} C_VEL
LIN {X 0,Y 214.085,Z 292.78,A -85,B 0,C 180,E1 -20739.65,E2 -20739.65} C_VEL
LIN {X 0,Y 215.583,Z 295.396,A -85,B 0,C 180,E1 -20740.285,E2 -20740.285} C_VEL
LIN {X 0,Y 217.321,Z 297.138,A -85,B 0,C 180,E1 -20740.91,E2 -20740.91} C_VEL
LIN {X 0,Y 219.612,Z 300.562,A -85,B 0,C 180,E1 -20741.762,E2 -20741.762} C_VEL
LIN {X 0,Y 220.941,Z 302.196,A -85,B 0,C 180,E1 -20742.226,E2 -20742.226} C_VEL
LIN {X 0,Y 227.078,Z 311.109,A -85,B 0,C 180,E1 -20744.308,E2 -20744.308} C_VEL
LIN {X 0,Y 234.077,Z 323.358,A -85,B 0,C 180,E1 -20746.552,E2 -20746.552} C_VEL
LIN {X 0,Y 239.802,Z 334.559,A -85,B 0,C 180,E1 -20748.28,E2 -20748.28} C_VEL
LIN {X 0,Y 246.697,Z 350.232,A -85,B 0,C 180,E1 -20750.281,E2 -20750.281} C_VEL
LIN {X 0,Y 247.397,Z 351.987,A -85,B 0,C 180,E1 -20750.481,E2 -20750.481} C_VEL
LIN {X 0,Y 244.411,Z 412.875,A -85,B 0,C 180,E1 -20752.157,E2 -20752.157} C_VEL
LIN {X 0,Y 243.295,Z 430.352,A -85,B 0,C 180,E1 -20752.72,E2 -20752.72} C_VEL
LIN {X 0,Y 241.557,Z 444.507,A -85,B 0,C 180,E1 -20753.45,E2 -20753.45} C_VEL
LIN {X 0,Y 239.225,Z 458.747,A -85,B 0,C 180,E1 -20754.535,E2 -20754.535} C_VEL
LIN {X 0,Y 236.528,Z 471.781,A -85,B 0,C 180,E1 -20755.887,E2 -20755.887} C_VEL
LIN {X 0,Y 233.567,Z 484.138,A -85,B 0,C 180,E1 -20757.562,E2 -20757.562} C_VEL
LIN {X 0,Y 230.275,Z 495.654,A -85,B 0,C 180,E1 -20759.51,E2 -20759.51} C_VEL
LIN {X 0,Y 226.706,Z 506.49,A -85,B 0,C 180,E1 -20761.787,E2 -20761.787} C_VEL
LIN {X 0,Y 223.353,Z 516.242,A -85,B 0,C 180,E1 -20764.364,E2 -20764.364} C_VEL
LIN {X 0,Y 220.312,Z 524.332,A -85,B 0,C 180,E1 -20766.998,E2 -20766.998} C_VEL
LIN {X 0,Y 217.889,Z 531.07,A -85,B 0,C 180,E1 -20769.712,E2 -20769.712} C_VEL
LIN {X 0,Y 215.578,Z 537.482,A -85,B 0,C 180,E1 -20772.938,E2 -20772.938} C_VEL
LIN {X 0,Y 213.919,Z 541.929,A -85,B 0,C 180,E1 -20775.735,E2 -20775.735} C_VEL
LIN {X 0,Y 212.785,Z 545.418,A -85,B 0,C 180,E1 -20778.57,E2 -20778.57} C_VEL
LIN {X 0,Y 211.882,Z 548.818,A -85,B 0,C 180,E1 -20782.376,E2 -20782.376} C_VEL
LIN {X 0,Y 211.442,Z 550.834,A -85,B 0,C 180,E1 -20786.188,E2 -20786.188} C_VEL
LIN {X 0,Y 211.438,Z 551.521,A -85,B 0,C 180,E1 -20790,E2 -20790} C_VEL
LIN {X 0,Y 211.442,Z 550.888,A -85,B 0,C 180,E1 -20793.811,E2 -20793.811} C_VEL
LIN {X 0,Y 211.88,Z 548.919,A -85,B 0,C 180,E1 -20797.624,E2 -20797.624} C_VEL
LIN {X 0,Y 212.764,Z 545.569,A -85,B 0,C 180,E1 -20801.431,E2 -20801.431} C_VEL
LIN {X 0,Y 214.336,Z 540.737,A -85,B 0,C 180,E1 -20805.207,E2 -20805.207} C_VEL
LIN {X 0,Y 216.177,Z 536.07,A -85,B 0,C 180,E1 -20807.989,E2 -20807.989} C_VEL
LIN {X 0,Y 218.418,Z 529.626,A -85,B 0,C 180,E1 -20811.072,E2 -20811.072} C_VEL
LIN {X 0,Y 221.2,Z 522.211,A -85,B 0,C 180,E1 -20813.896,E2 -20813.896} C_VEL
LIN {X 0,Y 224.33,Z 513.686,A -85,B 0,C 180,E1 -20816.514,E2 -20816.514} C_VEL
LIN {X 0,Y 227.842,Z 503.353,A -85,B 0,C 180,E1 -20819.066,E2 -20819.066} C_VEL
LIN {X 0,Y 231.164,Z 492.965,A -85,B 0,C 180,E1 -20821.12,E2 -20821.12} C_VEL
LIN {X 0,Y 234.259,Z 481.666,A -85,B 0,C 180,E1 -20822.94,E2 -20822.94} C_VEL
LIN {X 0,Y 237.181,Z 469.314,A -85,B 0,C 180,E1 -20824.519,E2 -20824.519} C_VEL
LIN {X 0,Y 239.925,Z 455.532,A -85,B 0,C 180,E1 -20825.862,E2 -20825.862} C_VEL
LIN {X 0,Y 242.09,Z 441.678,A -85,B 0,C 180,E1 -20826.845,E2 -20826.845} C_VEL
LIN {X 0,Y 243.615,Z 427.042,A -85,B 0,C 180,E1 -20827.559,E2 -20827.559} C_VEL
LIN {X 0,Y 246.009,Z 384.49,A -85,B 0,C 180,E1 -20828.734,E2 -20828.734} C_VEL
LIN {X 0,Y 247.533,Z 352.202,A -85,B 0,C 180,E1 -20829.634,E2 -20829.634} C_VEL
LIN {X 0,Y 241.623,Z 338.384,A -85,B 0,C 180,E1 -20831.34,E2 -20831.34} C_VEL
LIN {X 0,Y 235.334,Z 325.565,A -85,B 0,C 180,E1 -20833.228,E2 -20833.228} C_VEL
LIN {X 0,Y 228.55,Z 313.522,A -85,B 0,C 180,E1 -20835.376,E2 -20835.376} C_VEL
LIN {X 0,Y 225.357,Z 308.522,A -85,B 0,C 180,E1 -20836.432,E2 -20836.432} C_VEL
LIN {X 0,Y 222.56,Z 304.575,A -85,B 0,C 180,E1 -20837.38,E2 -20837.38} C_VEL
LIN {X 0,Y 219.925,Z 300.874,A -85,B 0,C 180,E1 -20838.31,E2 -20838.31} C_VEL
LIN {X 0,Y 217.611,Z 297.722,A -85,B 0,C 180,E1 -20839.156,E2 -20839.156} C_VEL
LIN {X 0,Y 216.866,Z 296.502,A -85,B 0,C 180,E1 -20839.445,E2 -20839.445} C_VEL
LIN {X 0,Y 214.64,Z 294.096,A -85,B 0,C 180,E1 -20840.269,E2 -20840.269} C_VEL
LIN {X 0,Y 213.849,Z 292.015,A -85,B 0,C 180,E1 -20840.793,E2 -20840.793} C_VEL
LIN {X 0,Y 213.755,Z 291.517,A -85,B 0,C 180,E1 -20841.34,E2 -20841.34} C_VEL
LIN {X 0,Y 213.765,Z 291.418,A -85,B 0,C 180,E1 -20846.019,E2 -20846.019} C_VEL
LIN {X 0,Y 213.778,Z 291.472,A -85,B 0,C 180,E1 -20850.453,E2 -20850.453} C_VEL
LIN {X 0,Y 213.798,Z 291.462,A -85,B 0,C 180,E1 -20854.701,E2 -20854.701} C_VEL
LIN {X 0,Y 213.808,Z 291.456,A -85,B 0,C 180,E1 -20858.803,E2 -20858.803} C_VEL
LIN {X 0,Y 213.94,Z 291.457,A -85,B 0,C 180,E1 -20862.803,E2 -20862.803} C_VEL
LIN {X 0,Y 213.947,Z 291.446,A -85,B 0,C 180,E1 -20866.706,E2 -20866.706} C_VEL
LIN {X 0,Y 214.137,Z 291.411,A -85,B 0,C 180,E1 -20870.555,E2 -20870.555} C_VEL
LIN {X 0,Y 214.097,Z 291.442,A -85,B 0,C 180,E1 -20874.348,E2 -20874.348} C_VEL
LIN {X 0,Y 214.441,Z 291.371,A -85,B 0,C 180,E1 -20878.122,E2 -20878.122} C_VEL
LIN {X 0,Y 214.55,Z 291.38,A -85,B 0,C 180,E1 -20880,E2 -20880} C_VEL
LIN {X 0,Y 214.44,Z 291.389,A -85,B 0,C 180,E1 -20881.878,E2 -20881.878} C_VEL
LIN {X 0,Y 214.236,Z 291.423,A -85,B 0,C 180,E1 -20887.54,E2 -20887.54} C_VEL
LIN {X 0,Y 214.04,Z 291.426,A -85,B 0,C 180,E1 -20891.362,E2 -20891.362} C_VEL
LIN {X 0,Y 213.924,Z 291.445,A -85,B 0,C 180,E1 -20895.237,E2 -20895.237} C_VEL
LIN {X 0,Y 213.864,Z 291.471,A -85,B 0,C 180,E1 -20899.185,E2 -20899.185} C_VEL
LIN {X 0,Y 213.843,Z 291.456,A -85,B 0,C 180,E1 -20903.227,E2 -20903.227} C_VEL
LIN {X 0,Y 213.826,Z 291.456,A -85,B 0,C 180,E1 -20907.45,E2 -20907.45} C_VEL
LIN {X 0,Y 213.773,Z 291.443,A -85,B 0,C 180,E1 -20911.736,E2 -20911.736} C_VEL
LIN {X 0,Y 213.753,Z 291.418,A -85,B 0,C 180,E1 -20914.021,E2 -20914.021} C_VEL
LIN {X 0,Y 213.691,Z 291.867,A -85,B 0,C 180,E1 -20915.053,E2 -20915.053} C_VEL
LIN {X 0,Y 213.528,Z 293.875,A -85,B 0,C 180,E1 -20916.526,E2 -20916.526} C_VEL
LIN {X 0,Y 213.632,Z 298.164,A -85,B 0,C 180,E1 -20918.309,E2 -20918.309} C_VEL
LIN {X 0,Y 214.74,Z 303.429,A -85,B 0,C 180,E1 -20919.908,E2 -20919.908} C_VEL
LIN {X 0,Y 216.74,Z 307.43,A -85,B 0,C 180,E1 -20920.972,E2 -20920.972} C_VEL
LIN {X 0,Y 221.847,Z 315.547,A -85,B 0,C 180,E1 -20922.846,E2 -20922.846} C_VEL
LIN {X 0,Y 228.195,Z 326.714,A -85,B 0,C 180,E1 -20925.024,E2 -20925.024} C_VEL
LIN {X 0,Y 234.99,Z 340.482,A -85,B 0,C 180,E1 -20927.217,E2 -20927.217} C_VEL
LIN {X 0,Y 241.869,Z 356.807,A -85,B 0,C 180,E1 -20929.334,E2 -20929.334} C_VEL
LIN {X 0,Y 238.09,Z 429.236,A -85,B 0,C 180,E1 -20931.385,E2 -20931.385} C_VEL
LIN {X 0,Y 236.561,Z 443.18,A -85,B 0,C 180,E1 -20932.01,E2 -20932.01} C_VEL
LIN {X 0,Y 234.462,Z 456.462,A -85,B 0,C 180,E1 -20932.898,E2 -20932.898} C_VEL
LIN {X 0,Y 231.934,Z 469.073,A -85,B 0,C 180,E1 -20934.05,E2 -20934.05} C_VEL
LIN {X 0,Y 228.726,Z 482.183,A -85,B 0,C 180,E1 -20935.626,E2 -20935.626} C_VEL
LIN {X 0,Y 225.272,Z 494.521,A -85,B 0,C 180,E1 -20937.548,E2 -20937.548} C_VEL
LIN {X 0,Y 221.953,Z 504.894,A -85,B 0,C 180,E1 -20939.561,E2 -20939.561} C_VEL
LIN {X 0,Y 218.117,Z 515.61,A -85,B 0,C 180,E1 -20942.148,E2 -20942.148} C_VEL
LIN {X 0,Y 214.772,Z 524.458,A -85,B 0,C 180,E1 -20944.825,E2 -20944.825} C_VEL
LIN {X 0,Y 211.977,Z 531.821,A -85,B 0,C 180,E1 -20947.588,E2 -20947.588} C_VEL
LIN {X 0,Y 209.712,Z 537.961,A -85,B 0,C 180,E1 -20950.42,E2 -20950.42} C_VEL
LIN {X 0,Y 207.199,Z 544.482,A -85,B 0,C 180,E1 -20954.256,E2 -20954.256} C_VEL
LIN {X 0,Y 205.519,Z 549.362,A -85,B 0,C 180,E1 -20958.16,E2 -20958.16} C_VEL
LIN {X 0,Y 204.635,Z 552.756,A -85,B 0,C 180,E1 -20962.104,E2 -20962.104} C_VEL
LIN {X 0,Y 204.258,Z 554.814,A -85,B 0,C 180,E1 -20966.213,E2 -20966.213} C_VEL
LIN {X 0,Y 204.337,Z 555.42,A -85,B 0,C 180,E1 -20970,E2 -20970} C_VEL
LIN {X 0,Y 204.26,Z 554.742,A -85,B 0,C 180,E1 -20973.946,E2 -20973.946} C_VEL
LIN {X 0,Y 204.636,Z 552.721,A -85,B 0,C 180,E1 -20977.896,E2 -20977.896} C_VEL
LIN {X 0,Y 205.522,Z 549.309,A -85,B 0,C 180,E1 -20981.84,E2 -20981.84} C_VEL
LIN {X 0,Y 207.198,Z 544.404,A -85,B 0,C 180,E1 -20985.745,E2 -20985.745} C_VEL
LIN {X 0,Y 209.621,Z 537.862,A -85,B 0,C 180,E1 -20989.589,E2 -20989.589} C_VEL
LIN {X 0,Y 212.344,Z 530.582,A -85,B 0,C 180,E1 -20992.885,E2 -20992.885} C_VEL
LIN {X 0,Y 215.851,Z 521.564,A -85,B 0,C 180,E1 -20996.075,E2 -20996.075} C_VEL
LIN {X 0,Y 219.277,Z 512.103,A -85,B 0,C 180,E1 -20998.735,E2 -20998.735} C_VEL
LIN {X 0,Y 223.016,Z 501.63,A -85,B 0,C 180,E1 -21001.066,E2 -21001.066} C_VEL
LIN {X 0,Y 226.415,Z 490.25,A -85,B 0,C 180,E1 -21003.129,E2 -21003.129} C_VEL
LIN {X 0,Y 229.512,Z 478.818,A -85,B 0,C 180,E1 -21004.772,E2 -21004.772} C_VEL
LIN {X 0,Y 232.344,Z 466.677,A -85,B 0,C 180,E1 -21006.145,E2 -21006.145} C_VEL
LIN {X 0,Y 234.935,Z 453.311,A -85,B 0,C 180,E1 -21007.284,E2 -21007.284} C_VEL
LIN {X 0,Y 236.921,Z 438.709,A -85,B 0,C 180,E1 -21008.192,E2 -21008.192} C_VEL
LIN {X 0,Y 238.161,Z 426.209,A -85,B 0,C 180,E1 -21008.676,E2 -21008.676} C_VEL
LIN {X 0,Y 241.758,Z 357.856,A -85,B 0,C 180,E1 -21010.586,E2 -21010.586} C_VEL
LIN {X 0,Y 241.535,Z 356.2,A -85,B 0,C 180,E1 -21010.695,E2 -21010.695} C_VEL
LIN {X 0,Y 236.369,Z 343.702,A -85,B 0,C 180,E1 -21012.277,E2 -21012.277} C_VEL
LIN {X 0,Y 229.376,Z 329.123,A -85,B 0,C 180,E1 -21014.504,E2 -21014.504} C_VEL
LIN {X 0,Y 222.361,Z 316.479,A -85,B 0,C 180,E1 -21016.884,E2 -21016.884} C_VEL
LIN {X 0,Y 216.446,Z 307.028,A -85,B 0,C 180,E1 -21019.044,E2 -21019.044} C_VEL
LIN {X 0,Y 213.082,Z 301.958,A -85,B 0,C 180,E1 -21020.355,E2 -21020.355} C_VEL
LIN {X 0,Y 210.652,Z 298.525,A -85,B 0,C 180,E1 -21021.34,E2 -21021.34} C_VEL
LIN {X 0,Y 209.942,Z 297.529,A -85,B 0,C 180,E1 -21021.636,E2 -21021.636} C_VEL
LIN {X 0,Y 207.696,Z 295.177,A -85,B 0,C 180,E1 -21022.553,E2 -21022.553} C_VEL
LIN {X 0,Y 206.802,Z 293.053,A -85,B 0,C 180,E1 -21023.128,E2 -21023.128} C_VEL
LIN {X 0,Y 206.729,Z 292.384,A -85,B 0,C 180,E1 -21023.794,E2 -21023.794} C_VEL
LIN {X 0,Y 206.723,Z 292.319,A -85,B 0,C 180,E1 -21028.202,E2 -21028.202} C_VEL
LIN {X 0,Y 206.764,Z 292.335,A -85,B 0,C 180,E1 -21032.096,E2 -21032.096} C_VEL
LIN {X 0,Y 206.783,Z 292.336,A -85,B 0,C 180,E1 -21036.584,E2 -21036.584} C_VEL
LIN {X 0,Y 206.873,Z 292.323,A -85,B 0,C 180,E1 -21042.197,E2 -21042.197} C_VEL
LIN {X 0,Y 206.907,Z 292.337,A -85,B 0,C 180,E1 -21046.245,E2 -21046.245} C_VEL
LIN {X 0,Y 207.102,Z 292.287,A -85,B 0,C 180,E1 -21050.231,E2 -21050.231} C_VEL
LIN {X 0,Y 207.174,Z 292.3,A -85,B 0,C 180,E1 -21052.201,E2 -21052.201} C_VEL
LIN {X 0,Y 207.378,Z 292.267,A -85,B 0,C 180,E1 -21058.058,E2 -21058.058} C_VEL
LIN {X 0,Y 207.511,Z 292.256,A -85,B 0,C 180,E1 -21060,E2 -21060} C_VEL
LIN {X 0,Y 207.378,Z 292.25,A -85,B 0,C 180,E1 -21061.942,E2 -21061.942} C_VEL
LIN {X 0,Y 207.137,Z 292.285,A -85,B 0,C 180,E1 -21067.8,E2 -21067.8} C_VEL
LIN {X 0,Y 206.928,Z 292.334,A -85,B 0,C 180,E1 -21071.758,E2 -21071.758} C_VEL
LIN {X 0,Y 206.861,Z 292.319,A -85,B 0,C 180,E1 -21075.771,E2 -21075.771} C_VEL
LIN {X 0,Y 206.78,Z 292.334,A -85,B 0,C 180,E1 -21079.87,E2 -21079.87} C_VEL
LIN {X 0,Y 206.761,Z 292.353,A -85,B 0,C 180,E1 -21084.073,E2 -21084.073} C_VEL
LIN {X 0,Y 206.742,Z 292.355,A -85,B 0,C 180,E1 -21088.419,E2 -21088.419} C_VEL
LIN {X 0,Y 206.707,Z 292.292,A -85,B 0,C 180,E1 -21092.956,E2 -21092.956} C_VEL
LIN {X 0,Y 206.737,Z 292.497,A -85,B 0,C 180,E1 -21096.657,E2 -21096.657} C_VEL
LIN {X 0,Y 206.95,Z 293.516,A -85,B 0,C 180,E1 -21097.222,E2 -21097.222} C_VEL
LIN {X 0,Y 208.567,Z 296.316,A -85,B 0,C 180,E1 -21097.997,E2 -21097.997} C_VEL
LIN {X 0,Y 210.5,Z 298.086,A -85,B 0,C 180,E1 -21098.762,E2 -21098.762} C_VEL
LIN {X 0,Y 212.666,Z 301.437,A -85,B 0,C 180,E1 -21099.66,E2 -21099.66} C_VEL
LIN {X 0,Y 214.143,Z 303.198,A -85,B 0,C 180,E1 -21100.226,E2 -21100.226} C_VEL
LIN {X 0,Y 218.03,Z 308.66,A -85,B 0,C 180,E1 -21101.689,E2 -21101.689} C_VEL
LIN {X 0,Y 222.994,Z 315.785,A -85,B 0,C 180,E1 -21103.434,E2 -21103.434} C_VEL
LIN {X 0,Y 229.856,Z 328.048,A -85,B 0,C 180,E1 -21105.744,E2 -21105.744} C_VEL
LIN {X 0,Y 235.842,Z 340.049,A -85,B 0,C 180,E1 -21107.636,E2 -21107.636} C_VEL
LIN {X 0,Y 241.842,Z 354.083,A -85,B 0,C 180,E1 -21109.464,E2 -21109.464} C_VEL
LIN {X 0,Y 238.899,Z 411.973,A -85,B 0,C 180,E1 -21111.085,E2 -21111.085} C_VEL
LIN {X 0,Y 237.675,Z 430.434,A -85,B 0,C 180,E1 -21111.682,E2 -21111.682} C_VEL
LIN {X 0,Y 235.892,Z 444.584,A -85,B 0,C 180,E1 -21112.423,E2 -21112.423} C_VEL
LIN {X 0,Y 233.475,Z 458.82,A -85,B 0,C 180,E1 -21113.523,E2 -21113.523} C_VEL
LIN {X 0,Y 230.686,Z 471.851,A -85,B 0,C 180,E1 -21114.898,E2 -21114.898} C_VEL
LIN {X 0,Y 227.58,Z 484.209,A -85,B 0,C 180,E1 -21116.599,E2 -21116.599} C_VEL
LIN {X 0,Y 224.183,Z 495.724,A -85,B 0,C 180,E1 -21118.589,E2 -21118.589} C_VEL
LIN {X 0,Y 220.456,Z 506.559,A -85,B 0,C 180,E1 -21120.912,E2 -21120.912} C_VEL
LIN {X 0,Y 216.941,Z 516.311,A -85,B 0,C 180,E1 -21123.549,E2 -21123.549} C_VEL
LIN {X 0,Y 213.754,Z 524.401,A -85,B 0,C 180,E1 -21126.249,E2 -21126.249} C_VEL
LIN {X 0,Y 211.367,Z 530.645,A -85,B 0,C 180,E1 -21128.806,E2 -21128.806} C_VEL
LIN {X 0,Y 208.783,Z 537.55,A -85,B 0,C 180,E1 -21132.365,E2 -21132.365} C_VEL
LIN {X 0,Y 206.998,Z 541.997,A -85,B 0,C 180,E1 -21135.248,E2 -21135.248} C_VEL
LIN {X 0,Y 205.819,Z 545.486,A -85,B 0,C 180,E1 -21138.178,E2 -21138.178} C_VEL
LIN {X 0,Y 204.845,Z 548.885,A -85,B 0,C 180,E1 -21142.112,E2 -21142.112} C_VEL
LIN {X 0,Y 204.366,Z 550.901,A -85,B 0,C 180,E1 -21146.056,E2 -21146.056} C_VEL
LIN {X 0,Y 204.343,Z 551.587,A -85,B 0,C 180,E1 -21150,E2 -21150} C_VEL
LIN {X 0,Y 204.366,Z 550.954,A -85,B 0,C 180,E1 -21153.944,E2 -21153.944} C_VEL
LIN {X 0,Y 204.843,Z 548.985,A -85,B 0,C 180,E1 -21157.888,E2 -21157.888} C_VEL
LIN {X 0,Y 205.794,Z 545.635,A -85,B 0,C 180,E1 -21161.823,E2 -21161.823} C_VEL
LIN {X 0,Y 207.47,Z 540.803,A -85,B 0,C 180,E1 -21165.723,E2 -21165.723} C_VEL
LIN {X 0,Y 209.403,Z 536.136,A -85,B 0,C 180,E1 -21168.592,E2 -21168.592} C_VEL
LIN {X 0,Y 211.57,Z 530.194,A -85,B 0,C 180,E1 -21171.547,E2 -21171.547} C_VEL
LIN {X 0,Y 214.694,Z 522.275,A -85,B 0,C 180,E1 -21174.668,E2 -21174.668} C_VEL
LIN {X 0,Y 217.972,Z 513.751,A -85,B 0,C 180,E1 -21177.351,E2 -21177.351} C_VEL
LIN {X 0,Y 221.653,Z 503.416,A -85,B 0,C 180,E1 -21179.959,E2 -21179.959} C_VEL
LIN {X 0,Y 225.105,Z 493.028,A -85,B 0,C 180,E1 -21182.056,E2 -21182.056} C_VEL
LIN {X 0,Y 228.34,Z 481.728,A -85,B 0,C 180,E1 -21183.907,E2 -21183.907} C_VEL
LIN {X 0,Y 231.379,Z 469.375,A -85,B 0,C 180,E1 -21185.514,E2 -21185.514} C_VEL
LIN {X 0,Y 234.221,Z 455.591,A -85,B 0,C 180,E1 -21186.877,E2 -21186.877} C_VEL
LIN {X 0,Y 236.461,Z 441.735,A -85,B 0,C 180,E1 -21187.874,E2 -21187.874} C_VEL
LIN {X 0,Y 238.01,Z 427.358,A -85,B 0,C 180,E1 -21188.588,E2 -21188.588} C_VEL
LIN {X 0,Y 240.543,Z 383.869,A -85,B 0,C 180,E1 -21189.812,E2 -21189.812} C_VEL
LIN {X 0,Y 241.995,Z 354.33,A -85,B 0,C 180,E1 -21190.648,E2 -21190.648} C_VEL
LIN {X 0,Y 235.908,Z 340.182,A -85,B 0,C 180,E1 -21192.502,E2 -21192.502} C_VEL
LIN {X 0,Y 230.629,Z 329.4,A -85,B 0,C 180,E1 -21194.175,E2 -21194.175} C_VEL
LIN {X 0,Y 224.172,Z 317.776,A -85,B 0,C 180,E1 -21196.33,E2 -21196.33} C_VEL
LIN {X 0,Y 221.372,Z 313.388,A -85,B 0,C 180,E1 -21197.301,E2 -21197.301} C_VEL
LIN {X 0,Y 216.253,Z 306.158,A -85,B 0,C 180,E1 -21199.153,E2 -21199.153} C_VEL
LIN {X 0,Y 213.204,Z 301.943,A -85,B 0,C 180,E1 -21200.329,E2 -21200.329} C_VEL
LIN {X 0,Y 211.031,Z 299.149,A -85,B 0,C 180,E1 -21201.195,E2 -21201.195} C_VEL
LIN {X 0,Y 210.174,Z 297.634,A -85,B 0,C 180,E1 -21201.569,E2 -21201.569} C_VEL
LIN {X 0,Y 207.845,Z 295.441,A -85,B 0,C 180,E1 -21202.508,E2 -21202.508} C_VEL
LIN {X 0,Y 206.797,Z 292.881,A -85,B 0,C 180,E1 -21203.203,E2 -21203.203} C_VEL
LIN {X 0,Y 206.71,Z 292.378,A -85,B 0,C 180,E1 -21203.791,E2 -21203.791} C_VEL
LIN {X 0,Y 206.726,Z 292.301,A -85,B 0,C 180,E1 -21208.201,E2 -21208.201} C_VEL
LIN {X 0,Y 206.764,Z 292.349,A -85,B 0,C 180,E1 -21212.096,E2 -21212.096} C_VEL
LIN {X 0,Y 206.782,Z 292.354,A -85,B 0,C 180,E1 -21216.583,E2 -21216.583} C_VEL
LIN {X 0,Y 206.87,Z 292.342,A -85,B 0,C 180,E1 -21222.196,E2 -21222.196} C_VEL
LIN {X 0,Y 206.89,Z 292.319,A -85,B 0,C 180,E1 -21226.244,E2 -21226.244} C_VEL
LIN {X 0,Y 207.096,Z 292.29,A -85,B 0,C 180,E1 -21230.231,E2 -21230.231} C_VEL
LIN {X 0,Y 207.058,Z 292.318,A -85,B 0,C 180,E1 -21234.155,E2 -21234.155} C_VEL
LIN {X 0,Y 207.377,Z 292.25,A -85,B 0,C 180,E1 -21238.058,E2 -21238.058} C_VEL
LIN {X 0,Y 207.514,Z 292.255,A -85,B 0,C 180,E1 -21240,E2 -21240} C_VEL
LIN {X 0,Y 207.079,Z 292.287,A -85,B 0,C 180,E1 -21243.892,E2 -21243.892} C_VEL
LIN {X 0,Y 207.173,Z 292.3,A -85,B 0,C 180,E1 -21247.799,E2 -21247.799} C_VEL
LIN {X 0,Y 206.976,Z 292.309,A -85,B 0,C 180,E1 -21251.755,E2 -21251.755} C_VEL
LIN {X 0,Y 206.859,Z 292.32,A -85,B 0,C 180,E1 -21255.771,E2 -21255.771} C_VEL
LIN {X 0,Y 206.795,Z 292.348,A -85,B 0,C 180,E1 -21259.868,E2 -21259.868} C_VEL
LIN {X 0,Y 206.76,Z 292.347,A -85,B 0,C 180,E1 -21264.072,E2 -21264.072} C_VEL
LIN {X 0,Y 206.741,Z 292.342,A -85,B 0,C 180,E1 -21268.419,E2 -21268.419} C_VEL
LIN {X 0,Y 206.699,Z 292.303,A -85,B 0,C 180,E1 -21272.958,E2 -21272.958} C_VEL
LIN {X 0,Y 206.731,Z 292.467,A -85,B 0,C 180,E1 -21276.356,E2 -21276.356} C_VEL
LIN {X 0,Y 206.932,Z 293.51,A -85,B 0,C 180,E1 -21276.921,E2 -21276.921} C_VEL
LIN {X 0,Y 208.357,Z 296.117,A -85,B 0,C 180,E1 -21277.626,E2 -21277.626} C_VEL
LIN {X 0,Y 210.474,Z 298.13,A -85,B 0,C 180,E1 -21278.474,E2 -21278.474} C_VEL
LIN {X 0,Y 212.725,Z 301.49,A -85,B 0,C 180,E1 -21279.405,E2 -21279.405} C_VEL
LIN {X 0,Y 215.165,Z 305.06,A -85,B 0,C 180,E1 -21280.368,E2 -21280.368} C_VEL
LIN {X 0,Y 216.74,Z 307.43,A -85,B 0,C 180,E1 -21280.972,E2 -21280.972} C_VEL
LIN {X 0,Y 218.065,Z 310.547,A -85,B 0,C 180,E1 -21281.523,E2 -21281.523} C_VEL
LIN {X 0,Y 219.018,Z 316.892,A -85,B 0,C 180,E1 -21282.108,E2 -21282.108} C_VEL
LIN {X 0,Y 219.989,Z 323.242,A -85,B 0,C 180,E1 -21282.686,E2 -21282.686} C_VEL
LIN {X 0,Y 221.37,Z 326.367,A -85,B 0,C 180,E1 -21283.217,E2 -21283.217} C_VEL
LIN {X 0,Y 227.676,Z 338.699,A -85,B 0,C 180,E1 -21285.415,E2 -21285.415} C_VEL
LIN {X 0,Y 233.271,Z 351.195,A -85,B 0,C 180,E1 -21287.267,E2 -21287.267} C_VEL
LIN {X 0,Y 236.407,Z 358.924,A -85,B 0,C 180,E1 -21288.273,E2 -21288.273} C_VEL
LIN {X 0,Y 232.644,Z 428.673,A -85,B 0,C 180,E1 -21290.282,E2 -21290.282} C_VEL
LIN {X 0,Y 231.017,Z 443.124,A -85,B 0,C 180,E1 -21290.929,E2 -21290.929} C_VEL
LIN {X 0,Y 228.845,Z 456.403,A -85,B 0,C 180,E1 -21291.827,E2 -21291.827} C_VEL
LIN {X 0,Y 226.227,Z 469.012,A -85,B 0,C 180,E1 -21292.994,E2 -21292.994} C_VEL
LIN {X 0,Y 222.882,Z 482.121,A -85,B 0,C 180,E1 -21294.592,E2 -21294.592} C_VEL
LIN {X 0,Y 219.256,Z 494.458,A -85,B 0,C 180,E1 -21296.543,E2 -21296.543} C_VEL
LIN {X 0,Y 215.847,Z 504.83,A -85,B 0,C 180,E1 -21298.604,E2 -21298.604} C_VEL
LIN {X 0,Y 211.819,Z 515.545,A -85,B 0,C 180,E1 -21301.244,E2 -21301.244} C_VEL
LIN {X 0,Y 208.345,Z 524.393,A -85,B 0,C 180,E1 -21303.991,E2 -21303.991} C_VEL
LIN {X 0,Y 204.945,Z 532.874,A -85,B 0,C 180,E1 -21307.308,E2 -21307.308} C_VEL
LIN {X 0,Y 202.231,Z 539.708,A -85,B 0,C 180,E1 -21310.723,E2 -21310.723} C_VEL
LIN {X 0,Y 200.329,Z 544.416,A -85,B 0,C 180,E1 -21313.701,E2 -21313.701} C_VEL
LIN {X 0,Y 198.54,Z 549.296,A -85,B 0,C 180,E1 -21317.738,E2 -21317.738} C_VEL
LIN {X 0,Y 197.581,Z 552.689,A -85,B 0,C 180,E1 -21321.82,E2 -21321.82} C_VEL
LIN {X 0,Y 197.174,Z 554.694,A -85,B 0,C 180,E1 -21325.912,E2 -21325.912} C_VEL
LIN {X 0,Y 197.244,Z 555.354,A -85,B 0,C 180,E1 -21330,E2 -21330} C_VEL
LIN {X 0,Y 197.174,Z 554.675,A -85,B 0,C 180,E1 -21334.088,E2 -21334.088} C_VEL
LIN {X 0,Y 197.582,Z 552.654,A -85,B 0,C 180,E1 -21338.18,E2 -21338.18} C_VEL
LIN {X 0,Y 198.543,Z 549.241,A -85,B 0,C 180,E1 -21342.262,E2 -21342.262} C_VEL
LIN {X 0,Y 200.327,Z 544.336,A -85,B 0,C 180,E1 -21346.299,E2 -21346.299} C_VEL
LIN {X 0,Y 202.883,Z 537.793,A -85,B 0,C 180,E1 -21350.267,E2 -21350.267} C_VEL
LIN {X 0,Y 205.781,Z 530.513,A -85,B 0,C 180,E1 -21353.659,E2 -21353.659} C_VEL
LIN {X 0,Y 209.46,Z 521.495,A -85,B 0,C 180,E1 -21356.934,E2 -21356.934} C_VEL
LIN {X 0,Y 213.076,Z 512.034,A -85,B 0,C 180,E1 -21359.653,E2 -21359.653} C_VEL
LIN {X 0,Y 216.955,Z 501.56,A -85,B 0,C 180,E1 -21362.035,E2 -21362.035} C_VEL
LIN {X 0,Y 220.66,Z 489.483,A -85,B 0,C 180,E1 -21364.258,E2 -21364.258} C_VEL
LIN {X 0,Y 224.108,Z 477.164,A -85,B 0,C 180,E1 -21366.014,E2 -21366.014} C_VEL
LIN {X 0,Y 227.083,Z 464.615,A -85,B 0,C 180,E1 -21367.399,E2 -21367.399} C_VEL
LIN {X 0,Y 229.74,Z 450.634,A -85,B 0,C 180,E1 -21368.556,E2 -21368.556} C_VEL
LIN {X 0,Y 231.671,Z 436.799,A -85,B 0,C 180,E1 -21369.361,E2 -21369.361} C_VEL
LIN {X 0,Y 232.876,Z 423.113,A -85,B 0,C 180,E1 -21369.864,E2 -21369.864} C_VEL
LIN {X 0,Y 236.344,Z 359.243,A -85,B 0,C 180,E1 -21371.661,E2 -21371.661} C_VEL
LIN {X 0,Y 232.587,Z 349.688,A -85,B 0,C 180,E1 -21372.88,E2 -21372.88} C_VEL
LIN {X 0,Y 226.301,Z 336.012,A -85,B 0,C 180,E1 -21374.969,E2 -21374.969} C_VEL
LIN {X 0,Y 220.13,Z 324.418,A -85,B 0,C 180,E1 -21377.132,E2 -21377.132} C_VEL
LIN {X 0,Y 215.563,Z 316.57,A -85,B 0,C 180,E1 -21378.839,E2 -21378.839} C_VEL
LIN {X 0,Y 209.789,Z 307.538,A -85,B 0,C 180,E1 -21381.151,E2 -21381.151} C_VEL
LIN {X 0,Y 206.64,Z 303.262,A -85,B 0,C 180,E1 -21382.482,E2 -21382.482} C_VEL
LIN {X 0,Y 204.277,Z 300.347,A -85,B 0,C 180,E1 -21383.52,E2 -21383.52} C_VEL
LIN {X 0,Y 203.283,Z 298.564,A -85,B 0,C 180,E1 -21384.004,E2 -21384.004} C_VEL
LIN {X 0,Y 200.817,Z 296.291,A -85,B 0,C 180,E1 -21385.119,E2 -21385.119} C_VEL
LIN {X 0,Y 199.744,Z 293.857,A -85,B 0,C 180,E1 -21385.872,E2 -21385.872} C_VEL
LIN {X 0,Y 199.666,Z 293.222,A -85,B 0,C 180,E1 -21386.783,E2 -21386.783} C_VEL
LIN {X 0,Y 199.71,Z 293.216,A -85,B 0,C 180,E1 -21391.613,E2 -21391.613} C_VEL
LIN {X 0,Y 199.735,Z 293.208,A -85,B 0,C 180,E1 -21397.229,E2 -21397.229} C_VEL
LIN {X 0,Y 199.835,Z 293.205,A -85,B 0,C 180,E1 -21401.722,E2 -21401.722} C_VEL
LIN {X 0,Y 199.842,Z 293.211,A -85,B 0,C 180,E1 -21405.749,E2 -21405.749} C_VEL
LIN {X 0,Y 200.067,Z 293.161,A -85,B 0,C 180,E1 -21409.884,E2 -21409.884} C_VEL
LIN {X 0,Y 200.033,Z 293.179,A -85,B 0,C 180,E1 -21413.95,E2 -21413.95} C_VEL
LIN {X 0,Y 200.317,Z 293.144,A -85,B 0,C 180,E1 -21417.99,E2 -21417.99} C_VEL
LIN {X 0,Y 200.475,Z 293.131,A -85,B 0,C 180,E1 -21420,E2 -21420} C_VEL
LIN {X 0,Y 200.023,Z 293.175,A -85,B 0,C 180,E1 -21424.03,E2 -21424.03} C_VEL
LIN {X 0,Y 200.085,Z 293.161,A -85,B 0,C 180,E1 -21428.077,E2 -21428.077} C_VEL
LIN {X 0,Y 199.875,Z 293.212,A -85,B 0,C 180,E1 -21432.179,E2 -21432.179} C_VEL
LIN {X 0,Y 199.8,Z 293.202,A -85,B 0,C 180,E1 -21436.344,E2 -21436.344} C_VEL
LIN {X 0,Y 199.697,Z 293.212,A -85,B 0,C 180,E1 -21440.606,E2 -21440.606} C_VEL
LIN {X 0,Y 199.67,Z 293.224,A -85,B 0,C 180,E1 -21444.985,E2 -21444.985} C_VEL
LIN {X 0,Y 199.673,Z 293.225,A -85,B 0,C 180,E1 -21449.523,E2 -21449.523} C_VEL
LIN {X 0,Y 199.663,Z 293.271,A -85,B 0,C 180,E1 -21453.746,E2 -21453.746} C_VEL
LIN {X 0,Y 199.825,Z 294.087,A -85,B 0,C 180,E1 -21454.432,E2 -21454.432} C_VEL
LIN {X 0,Y 201.256,Z 296.83,A -85,B 0,C 180,E1 -21455.269,E2 -21455.269} C_VEL
LIN {X 0,Y 203.591,Z 298.973,A -85,B 0,C 180,E1 -21456.316,E2 -21456.316} C_VEL
LIN {X 0,Y 205.635,Z 302.223,A -85,B 0,C 180,E1 -21457.271,E2 -21457.271} C_VEL
LIN {X 0,Y 207.506,Z 304.284,A -85,B 0,C 180,E1 -21458.06,E2 -21458.06} C_VEL
LIN {X 0,Y 210.362,Z 308.085,A -85,B 0,C 180,E1 -21459.248,E2 -21459.248} C_VEL
LIN {X 0,Y 217.463,Z 318.305,A -85,B 0,C 180,E1 -21461.989,E2 -21461.989} C_VEL
LIN {X 0,Y 221.148,Z 324.24,A -85,B 0,C 180,E1 -21463.319,E2 -21463.319} C_VEL
LIN {X 0,Y 228.63,Z 338.473,A -85,B 0,C 180,E1 -21465.893,E2 -21465.893} C_VEL
LIN {X 0,Y 234.818,Z 352.458,A -85,B 0,C 180,E1 -21467.911,E2 -21467.911} C_VEL
LIN {X 0,Y 236.464,Z 356.827,A -85,B 0,C 180,E1 -21468.445,E2 -21468.445} C_VEL
LIN {X 0,Y 232.499,Z 426.834,A -85,B 0,C 180,E1 -21470.44,E2 -21470.44} C_VEL
LIN {X 0,Y 230.732,Z 441.616,A -85,B 0,C 180,E1 -21471.151,E2 -21471.151} C_VEL
LIN {X 0,Y 228.453,Z 455.516,A -85,B 0,C 180,E1 -21472.169,E2 -21472.169} C_VEL
LIN {X 0,Y 225.714,Z 468.456,A -85,B 0,C 180,E1 -21473.453,E2 -21473.453} C_VEL
LIN {X 0,Y 222.539,Z 481,A -85,B 0,C 180,E1 -21475.083,E2 -21475.083} C_VEL
LIN {X 0,Y 219.243,Z 492.435,A -85,B 0,C 180,E1 -21476.98,E2 -21476.98} C_VEL
LIN {X 0,Y 215.63,Z 502.935,A -85,B 0,C 180,E1 -21479.114,E2 -21479.114} C_VEL
LIN {X 0,Y 212.365,Z 511.738,A -85,B 0,C 180,E1 -21481.324,E2 -21481.324} C_VEL
LIN {X 0,Y 208.867,Z 520.61,A -85,B 0,C 180,E1 -21484.061,E2 -21484.061} C_VEL
LIN {X 0,Y 205.335,Z 529.106,A -85,B 0,C 180,E1 -21487.353,E2 -21487.353} C_VEL
LIN {X 0,Y 202.738,Z 535.944,A -85,B 0,C 180,E1 -21490.773,E2 -21490.773} C_VEL
LIN {X 0,Y 200.654,Z 540.665,A -85,B 0,C 180,E1 -21493.728,E2 -21493.728} C_VEL
LIN {X 0,Y 198.867,Z 545.553,A -85,B 0,C 180,E1 -21497.758,E2 -21497.758} C_VEL
LIN {X 0,Y 197.785,Z 548.953,A -85,B 0,C 180,E1 -21501.829,E2 -21501.829} C_VEL
LIN {X 0,Y 197.286,Z 550.968,A -85,B 0,C 180,E1 -21505.914,E2 -21505.914} C_VEL
LIN {X 0,Y 197.25,Z 551.654,A -85,B 0,C 180,E1 -21510,E2 -21510} C_VEL
LIN {X 0,Y 197.286,Z 551.021,A -85,B 0,C 180,E1 -21514.085,E2 -21514.085} C_VEL
LIN {X 0,Y 197.78,Z 549.052,A -85,B 0,C 180,E1 -21518.171,E2 -21518.171} C_VEL
LIN {X 0,Y 198.824,Z 545.701,A -85,B 0,C 180,E1 -21522.244,E2 -21522.244} C_VEL
LIN {X 0,Y 200.628,Z 540.868,A -85,B 0,C 180,E1 -21526.274,E2 -21526.274} C_VEL
LIN {X 0,Y 202.654,Z 536.201,A -85,B 0,C 180,E1 -21529.235,E2 -21529.235} C_VEL
LIN {X 0,Y 205.313,Z 529.418,A -85,B 0,C 180,E1 -21532.649,E2 -21532.649} C_VEL
LIN {X 0,Y 208.771,Z 520.991,A -85,B 0,C 180,E1 -21535.952,E2 -21535.952} C_VEL
LIN {X 0,Y 212.293,Z 512.193,A -85,B 0,C 180,E1 -21538.686,E2 -21538.686} C_VEL
LIN {X 0,Y 215.527,Z 503.48,A -85,B 0,C 180,E1 -21540.902,E2 -21540.902} C_VEL
LIN {X 0,Y 219.116,Z 493.09,A -85,B 0,C 180,E1 -21543.042,E2 -21543.042} C_VEL
LIN {X 0,Y 222.475,Z 481.79,A -85,B 0,C 180,E1 -21544.929,E2 -21544.929} C_VEL
LIN {X 0,Y 225.632,Z 469.436,A -85,B 0,C 180,E1 -21546.562,E2 -21546.562} C_VEL
LIN {X 0,Y 228.587,Z 455.65,A -85,B 0,C 180,E1 -21547.944,E2 -21547.944} C_VEL
LIN {X 0,Y 230.787,Z 442.553,A -85,B 0,C 180,E1 -21548.907,E2 -21548.907} C_VEL
LIN {X 0,Y 232.42,Z 428.38,A -85,B 0,C 180,E1 -21549.636,E2 -21549.636} C_VEL
LIN {X 0,Y 234.259,Z 400.151,A -85,B 0,C 180,E1 -21550.461,E2 -21550.461} C_VEL
LIN {X 0,Y 236.536,Z 356.459,A -85,B 0,C 180,E1 -21551.71,E2 -21551.71} C_VEL
LIN {X 0,Y 230.564,Z 342.606,A -85,B 0,C 180,E1 -21553.631,E2 -21553.631} C_VEL
LIN {X 0,Y 225.428,Z 332.1,A -85,B 0,C 180,E1 -21555.356,E2 -21555.356} C_VEL
LIN {X 0,Y 218.758,Z 320.098,A -85,B 0,C 180,E1 -21557.727,E2 -21557.727} C_VEL
LIN {X 0,Y 212.872,Z 311.709,A -85,B 0,C 180,E1 -21559.932,E2 -21559.932} C_VEL
LIN {X 0,Y 209.604,Z 307.229,A -85,B 0,C 180,E1 -21561.248,E2 -21561.248} C_VEL
LIN {X 0,Y 206.805,Z 303.381,A -85,B 0,C 180,E1 -21562.44,E2 -21562.44} C_VEL
LIN {X 0,Y 204.32,Z 300.433,A -85,B 0,C 180,E1 -21563.528,E2 -21563.528} C_VEL
LIN {X 0,Y 203.334,Z 298.605,A -85,B 0,C 180,E1 -21564.014,E2 -21564.014} C_VEL
LIN {X 0,Y 200.879,Z 296.372,A -85,B 0,C 180,E1 -21565.128,E2 -21565.128} C_VEL
LIN {X 0,Y 199.738,Z 293.774,A -85,B 0,C 180,E1 -21565.937,E2 -21565.937} C_VEL
LIN {X 0,Y 199.674,Z 293.252,A -85,B 0,C 180,E1 -21566.52,E2 -21566.52} C_VEL
LIN {X 0,Y 199.672,Z 293.223,A -85,B 0,C 180,E1 -21570.477,E2 -21570.477} C_VEL
LIN {X 0,Y 199.669,Z 293.224,A -85,B 0,C 180,E1 -21575.015,E2 -21575.015} C_VEL
LIN {X 0,Y 199.696,Z 293.212,A -85,B 0,C 180,E1 -21579.394,E2 -21579.394} C_VEL
LIN {X 0,Y 199.799,Z 293.204,A -85,B 0,C 180,E1 -21583.656,E2 -21583.656} C_VEL
LIN {X 0,Y 199.874,Z 293.213,A -85,B 0,C 180,E1 -21587.82,E2 -21587.82} C_VEL
LIN {X 0,Y 200.085,Z 293.161,A -85,B 0,C 180,E1 -21591.923,E2 -21591.923} C_VEL
LIN {X 0,Y 200.317,Z 293.129,A -85,B 0,C 180,E1 -21597.989,E2 -21597.989} C_VEL
LIN {X 0,Y 200.478,Z 293.13,A -85,B 0,C 180,E1 -21600,E2 -21600} C_VEL
LIN {X 0,Y 200.024,Z 293.165,A -85,B 0,C 180,E1 -21604.029,E2 -21604.029} C_VEL
LIN {X 0,Y 200.115,Z 293.175,A -85,B 0,C 180,E1 -21608.075,E2 -21608.075} C_VEL
LIN {X 0,Y 199.908,Z 293.194,A -85,B 0,C 180,E1 -21612.177,E2 -21612.177} C_VEL
LIN {X 0,Y 199.798,Z 293.197,A -85,B 0,C 180,E1 -21616.344,E2 -21616.344} C_VEL
LIN {X 0,Y 199.82,Z 293.21,A -85,B 0,C 180,E1 -21618.454,E2 -21618.454} C_VEL
LIN {X 0,Y 199.733,Z 293.218,A -85,B 0,C 180,E1 -21623.817,E2 -21623.817} C_VEL
LIN {X 0,Y 199.709,Z 293.217,A -85,B 0,C 180,E1 -21628.387,E2 -21628.387} C_VEL
LIN {X 0,Y 199.665,Z 293.221,A -85,B 0,C 180,E1 -21633.217,E2 -21633.217} C_VEL
LIN {X 0,Y 199.735,Z 293.827,A -85,B 0,C 180,E1 -21633.997,E2 -21633.997} C_VEL
LIN {X 0,Y 201.131,Z 296.737,A -85,B 0,C 180,E1 -21634.911,E2 -21634.911} C_VEL
LIN {X 0,Y 203.574,Z 298.96,A -85,B 0,C 180,E1 -21636.013,E2 -21636.013} C_VEL
LIN {X 0,Y 205.606,Z 302.216,A -85,B 0,C 180,E1 -21636.969,E2 -21636.969} C_VEL
LIN {X 0,Y 207.53,Z 304.339,A -85,B 0,C 180,E1 -21637.786,E2 -21637.786} C_VEL
LIN {X 0,Y 211.395,Z 309.913,A -85,B 0,C 180,E1 -21639.408,E2 -21639.408} C_VEL
LIN {X 0,Y 217.492,Z 319.647,A -85,B 0,C 180,E1 -21641.795,E2 -21641.795} C_VEL
LIN {X 0,Y 221.37,Z 326.367,A -85,B 0,C 180,E1 -21643.217,E2 -21643.217} C_VEL
LIN {X 0,Y 222.938,Z 329.213,A -85,B 0,C 180,E1 -21643.774,E2 -21643.774} C_VEL
LIN {X 0,Y 224.519,Z 334.3,A -85,B 0,C 180,E1 -21644.42,E2 -21644.42} C_VEL
LIN {X 0,Y 227.377,Z 351.269,A -85,B 0,C 180,E1 -21645.885,E2 -21645.885} C_VEL
LIN {X 0,Y 228.494,Z 354.773,A -85,B 0,C 180,E1 -21646.305,E2 -21646.305} C_VEL
LIN {X 0,Y 231.042,Z 361.09,A -85,B 0,C 180,E1 -21647.167,E2 -21647.167} C_VEL
LIN {X 0,Y 227.119,Z 429.892,A -85,B 0,C 180,E1 -21649.18,E2 -21649.18} C_VEL
LIN {X 0,Y 225.437,Z 443.848,A -85,B 0,C 180,E1 -21649.841,E2 -21649.841} C_VEL
LIN {X 0,Y 223.298,Z 456.343,A -85,B 0,C 180,E1 -21650.699,E2 -21650.699} C_VEL
LIN {X 0,Y 220.59,Z 468.951,A -85,B 0,C 180,E1 -21651.883,E2 -21651.883} C_VEL
LIN {X 0,Y 217.124,Z 482.059,A -85,B 0,C 180,E1 -21653.505,E2 -21653.505} C_VEL
LIN {X 0,Y 213.718,Z 493.329,A -85,B 0,C 180,E1 -21655.297,E2 -21655.297} C_VEL
LIN {X 0,Y 209.797,Z 504.767,A -85,B 0,C 180,E1 -21657.59,E2 -21657.59} C_VEL
LIN {X 0,Y 205.6,Z 515.481,A -85,B 0,C 180,E1 -21660.288,E2 -21660.288} C_VEL
LIN {X 0,Y 201.959,Z 524.328,A -85,B 0,C 180,E1 -21663.104,E2 -21663.104} C_VEL
LIN {X 0,Y 198.8,Z 531.69,A -85,B 0,C 180,E1 -21666.013,E2 -21666.013} C_VEL
LIN {X 0,Y 196.264,Z 537.829,A -85,B 0,C 180,E1 -21669.018,E2 -21669.018} C_VEL
LIN {X 0,Y 193.486,Z 544.35,A -85,B 0,C 180,E1 -21673.108,E2 -21673.108} C_VEL
LIN {X 0,Y 191.577,Z 549.23,A -85,B 0,C 180,E1 -21677.285,E2 -21677.285} C_VEL
LIN {X 0,Y 190.528,Z 552.623,A -85,B 0,C 180,E1 -21681.515,E2 -21681.515} C_VEL
LIN {X 0,Y 190.088,Z 554.628,A -85,B 0,C 180,E1 -21685.76,E2 -21685.76} C_VEL
LIN {X 0,Y 190.152,Z 555.287,A -85,B 0,C 180,E1 -21690,E2 -21690} C_VEL
LIN {X 0,Y 190.088,Z 554.608,A -85,B 0,C 180,E1 -21694.241,E2 -21694.241} C_VEL
LIN {X 0,Y 190.529,Z 552.587,A -85,B 0,C 180,E1 -21698.485,E2 -21698.485} C_VEL
LIN {X 0,Y 191.579,Z 549.173,A -85,B 0,C 180,E1 -21702.715,E2 -21702.715} C_VEL
LIN {X 0,Y 193.484,Z 544.268,A -85,B 0,C 180,E1 -21706.893,E2 -21706.893} C_VEL
LIN {X 0,Y 196.173,Z 537.724,A -85,B 0,C 180,E1 -21710.993,E2 -21710.993} C_VEL
LIN {X 0,Y 199.258,Z 530.445,A -85,B 0,C 180,E1 -21714.483,E2 -21714.483} C_VEL
LIN {X 0,Y 203.12,Z 521.426,A -85,B 0,C 180,E1 -21717.846,E2 -21717.846} C_VEL
LIN {X 0,Y 206.935,Z 511.964,A -85,B 0,C 180,E1 -21720.626,E2 -21720.626} C_VEL
LIN {X 0,Y 210.958,Z 501.49,A -85,B 0,C 180,E1 -21723.06,E2 -21723.06} C_VEL
LIN {X 0,Y 214.718,Z 489.734,A -85,B 0,C 180,E1 -21725.274,E2 -21725.274} C_VEL
LIN {X 0,Y 218.387,Z 477.092,A -85,B 0,C 180,E1 -21727.113,E2 -21727.113} C_VEL
LIN {X 0,Y 221.485,Z 464.543,A -85,B 0,C 180,E1 -21728.515,E2 -21728.515} C_VEL
LIN {X 0,Y 224.225,Z 450.56,A -85,B 0,C 180,E1 -21729.688,E2 -21729.688} C_VEL
LIN {X 0,Y 226.24,Z 436.721,A -85,B 0,C 180,E1 -21730.498,E2 -21730.498} C_VEL
LIN {X 0,Y 227.468,Z 423.004,A -85,B 0,C 180,E1 -21731.012,E2 -21731.012} C_VEL
LIN {X 0,Y 230.931,Z 361.614,A -85,B 0,C 180,E1 -21732.766,E2 -21732.766} C_VEL
LIN {X 0,Y 230.194,Z 359.064,A -85,B 0,C 180,E1 -21733.041,E2 -21733.041} C_VEL
LIN {X 0,Y 224.018,Z 344.587,A -85,B 0,C 180,E1 -21735.17,E2 -21735.17} C_VEL
LIN {X 0,Y 217.405,Z 331.319,A -85,B 0,C 180,E1 -21737.578,E2 -21737.578} C_VEL
LIN {X 0,Y 211.622,Z 321.269,A -85,B 0,C 180,E1 -21739.829,E2 -21739.829} C_VEL
LIN {X 0,Y 206.612,Z 313.221,A -85,B 0,C 180,E1 -21741.94,E2 -21741.94} C_VEL
LIN {X 0,Y 203.554,Z 309.016,A -85,B 0,C 180,E1 -21743.292,E2 -21743.292} C_VEL
LIN {X 0,Y 200.959,Z 305.587,A -85,B 0,C 180,E1 -21744.498,E2 -21744.498} C_VEL
LIN {X 0,Y 199.866,Z 304.221,A -85,B 0,C 180,E1 -21745.022,E2 -21745.022} C_VEL
LIN {X 0,Y 197.46,Z 301.358,A -85,B 0,C 180,E1 -21746.212,E2 -21746.212} C_VEL
LIN {X 0,Y 196.43,Z 299.552,A -85,B 0,C 180,E1 -21746.78,E2 -21746.78} C_VEL
LIN {X 0,Y 193.966,Z 297.385,A -85,B 0,C 180,E1 -21748.052,E2 -21748.052} C_VEL
LIN {X 0,Y 192.727,Z 294.741,A -85,B 0,C 180,E1 -21748.997,E2 -21748.997} C_VEL
LIN {X 0,Y 192.626,Z 294.15,A -85,B 0,C 180,E1 -21749.793,E2 -21749.793} C_VEL
LIN {X 0,Y 192.594,Z 294.107,A -85,B 0,C 180,E1 -21754.031,E2 -21754.031} C_VEL
LIN {X 0,Y 192.703,Z 294.09,A -85,B 0,C 180,E1 -21756.348,E2 -21756.348} C_VEL
LIN {X 0,Y 192.779,Z 294.087,A -85,B 0,C 180,E1 -21761.414,E2 -21761.414} C_VEL
LIN {X 0,Y 192.848,Z 294.079,A -85,B 0,C 180,E1 -21767.37,E2 -21767.37} C_VEL
LIN {X 0,Y 193.065,Z 294.047,A -85,B 0,C 180,E1 -21771.628,E2 -21771.628} C_VEL
LIN {X 0,Y 193.259,Z 294.021,A -85,B 0,C 180,E1 -21777.916,E2 -21777.916} C_VEL
LIN {X 0,Y 193.439,Z 294.006,A -85,B 0,C 180,E1 -21780,E2 -21780} C_VEL
LIN {X 0,Y 192.969,Z 294.054,A -85,B 0,C 180,E1 -21784.177,E2 -21784.177} C_VEL
LIN {X 0,Y 193.033,Z 294.037,A -85,B 0,C 180,E1 -21788.374,E2 -21788.374} C_VEL
LIN {X 0,Y 192.801,Z 294.088,A -85,B 0,C 180,E1 -21792.634,E2 -21792.634} C_VEL
LIN {X 0,Y 192.754,Z 294.087,A -85,B 0,C 180,E1 -21796.959,E2 -21796.959} C_VEL
LIN {X 0,Y 192.633,Z 294.092,A -85,B 0,C 180,E1 -21801.398,E2 -21801.398} C_VEL
LIN {X 0,Y 192.662,Z 294.106,A -85,B 0,C 180,E1 -21804.225,E2 -21804.225} C_VEL
LIN {X 0,Y 192.629,Z 294.094,A -85,B 0,C 180,E1 -21809.7,E2 -21809.7} C_VEL
LIN {X 0,Y 192.692,Z 294.49,A -85,B 0,C 180,E1 -21811.01,E2 -21811.01} C_VEL
LIN {X 0,Y 193.052,Z 295.728,A -85,B 0,C 180,E1 -21811.555,E2 -21811.555} C_VEL
LIN {X 0,Y 194.769,Z 298.319,A -85,B 0,C 180,E1 -21812.563,E2 -21812.563} C_VEL
LIN {X 0,Y 196.727,Z 299.833,A -85,B 0,C 180,E1 -21813.547,E2 -21813.547} C_VEL
LIN {X 0,Y 198.779,Z 303.139,A -85,B 0,C 180,E1 -21814.639,E2 -21814.639} C_VEL
LIN {X 0,Y 200.822,Z 305.257,A -85,B 0,C 180,E1 -21815.604,E2 -21815.604} C_VEL
LIN {X 0,Y 203.28,Z 308.74,A -85,B 0,C 180,E1 -21816.766,E2 -21816.766} C_VEL
LIN {X 0,Y 204.662,Z 310.485,A -85,B 0,C 180,E1 -21817.381,E2 -21817.381} C_VEL
LIN {X 0,Y 208.666,Z 316.07,A -85,B 0,C 180,E1 -21819.102,E2 -21819.102} C_VEL
LIN {X 0,Y 215.144,Z 325.435,A -85,B 0,C 180,E1 -21821.649,E2 -21821.649} C_VEL
LIN {X 0,Y 222.141,Z 338.516,A -85,B 0,C 180,E1 -21824.244,E2 -21824.244} C_VEL
LIN {X 0,Y 227.532,Z 350.042,A -85,B 0,C 180,E1 -21826.122,E2 -21826.122} C_VEL
LIN {X 0,Y 231.025,Z 358.425,A -85,B 0,C 180,E1 -21827.301,E2 -21827.301} C_VEL
LIN {X 0,Y 227.503,Z 421.071,A -85,B 0,C 180,E1 -21829.102,E2 -21829.102} C_VEL
LIN {X 0,Y 226.124,Z 435.675,A -85,B 0,C 180,E1 -21829.696,E2 -21829.696} C_VEL
LIN {X 0,Y 224.043,Z 449.518,A -85,B 0,C 180,E1 -21830.565,E2 -21830.565} C_VEL
LIN {X 0,Y 221.351,Z 462.967,A -85,B 0,C 180,E1 -21831.748,E2 -21831.748} C_VEL
LIN {X 0,Y 218.384,Z 475.155,A -85,B 0,C 180,E1 -21833.175,E2 -21833.175} C_VEL
LIN {X 0,Y 215.196,Z 486.567,A -85,B 0,C 180,E1 -21834.889,E2 -21834.889} C_VEL
LIN {X 0,Y 211.447,Z 498,A -85,B 0,C 180,E1 -21837.026,E2 -21837.026} C_VEL
LIN {X 0,Y 207.427,Z 508.478,A -85,B 0,C 180,E1 -21839.455,E2 -21839.455} C_VEL
LIN {X 0,Y 203.694,Z 517.932,A -85,B 0,C 180,E1 -21842.239,E2 -21842.239} C_VEL
LIN {X 0,Y 199.769,Z 526.948,A -85,B 0,C 180,E1 -21845.584,E2 -21845.584} C_VEL
LIN {X 0,Y 196.71,Z 534.21,A -85,B 0,C 180,E1 -21849.067,E2 -21849.067} C_VEL
LIN {X 0,Y 194.549,Z 539.294,A -85,B 0,C 180,E1 -21852.118,E2 -21852.118} C_VEL
LIN {X 0,Y 192.728,Z 543.372,A -85,B 0,C 180,E1 -21855.211,E2 -21855.211} C_VEL
LIN {X 0,Y 191.233,Z 547.499,A -85,B 0,C 180,E1 -21859.412,E2 -21859.412} C_VEL
LIN {X 0,Y 190.426,Z 550.196,A -85,B 0,C 180,E1 -21863.643,E2 -21863.643} C_VEL
LIN {X 0,Y 190.135,Z 551.543,A -85,B 0,C 180,E1 -21867.882,E2 -21867.882} C_VEL
LIN {X 0,Y 190.159,Z 551.72,A -85,B 0,C 180,E1 -21870,E2 -21870} C_VEL
LIN {X 0,Y 190.2,Z 551.087,A -85,B 0,C 180,E1 -21874.238,E2 -21874.238} C_VEL
LIN {X 0,Y 190.736,Z 549.118,A -85,B 0,C 180,E1 -21878.475,E2 -21878.475} C_VEL
LIN {X 0,Y 191.851,Z 545.767,A -85,B 0,C 180,E1 -21882.697,E2 -21882.697} C_VEL
LIN {X 0,Y 193.811,Z 540.934,A -85,B 0,C 180,E1 -21886.863,E2 -21886.863} C_VEL
LIN {X 0,Y 195.918,Z 536.267,A -85,B 0,C 180,E1 -21889.924,E2 -21889.924} C_VEL
LIN {X 0,Y 198.745,Z 529.483,A -85,B 0,C 180,E1 -21893.441,E2 -21893.441} C_VEL
LIN {X 0,Y 202.398,Z 521.055,A -85,B 0,C 180,E1 -21896.833,E2 -21896.833} C_VEL
LIN {X 0,Y 206.084,Z 512.257,A -85,B 0,C 180,E1 -21899.635,E2 -21899.635} C_VEL
LIN {X 0,Y 209.463,Z 503.543,A -85,B 0,C 180,E1 -21901.9,E2 -21901.9} C_VEL
LIN {X 0,Y 213.686,Z 491.83,A -85,B 0,C 180,E1 -21904.315,E2 -21904.315} C_VEL
LIN {X 0,Y 217.07,Z 480.428,A -85,B 0,C 180,E1 -21906.218,E2 -21906.218} C_VEL
LIN {X 0,Y 220.407,Z 467.733,A -85,B 0,C 180,E1 -21907.865,E2 -21907.865} C_VEL
LIN {X 0,Y 223.264,Z 454.581,A -85,B 0,C 180,E1 -21909.162,E2 -21909.162} C_VEL
LIN {X 0,Y 225.549,Z 441.086,A -85,B 0,C 180,E1 -21910.135,E2 -21910.135} C_VEL
LIN {X 0,Y 227.184,Z 426.667,A -85,B 0,C 180,E1 -21910.851,E2 -21910.851} C_VEL
LIN {X 0,Y 229.871,Z 382.774,A -85,B 0,C 180,E1 -21912.115,E2 -21912.115} C_VEL
LIN {X 0,Y 231.161,Z 358.608,A -85,B 0,C 180,E1 -21912.822,E2 -21912.822} C_VEL
LIN {X 0,Y 224.472,Z 343.065,A -85,B 0,C 180,E1 -21915.114,E2 -21915.114} C_VEL
LIN {X 0,Y 216.943,Z 328.551,A -85,B 0,C 180,E1 -21917.848,E2 -21917.848} C_VEL
LIN {X 0,Y 212.611,Z 321.569,A -85,B 0,C 180,E1 -21919.511,E2 -21919.511} C_VEL
LIN {X 0,Y 206.437,Z 312.902,A -85,B 0,C 180,E1 -21922.042,E2 -21922.042} C_VEL
LIN {X 0,Y 203.599,Z 309.068,A -85,B 0,C 180,E1 -21923.301,E2 -21923.301} C_VEL
LIN {X 0,Y 200.889,Z 305.449,A -85,B 0,C 180,E1 -21924.571,E2 -21924.571} C_VEL
LIN {X 0,Y 200.072,Z 304.393,A -85,B 0,C 180,E1 -21924.967,E2 -21924.967} C_VEL
LIN {X 0,Y 197.529,Z 301.42,A -85,B 0,C 180,E1 -21926.225,E2 -21926.225} C_VEL
LIN {X 0,Y 196.51,Z 299.55,A -85,B 0,C 180,E1 -21926.795,E2 -21926.795} C_VEL
LIN {X 0,Y 194.114,Z 297.569,A -85,B 0,C 180,E1 -21928.029,E2 -21928.029} C_VEL
LIN {X 0,Y 192.72,Z 294.74,A -85,B 0,C 180,E1 -21929.072,E2 -21929.072} C_VEL
LIN {X 0,Y 192.626,Z 294.169,A -85,B 0,C 180,E1 -21929.793,E2 -21929.793} C_VEL
LIN {X 0,Y 192.594,Z 294.1,A -85,B 0,C 180,E1 -21934.03,E2 -21934.03} C_VEL
LIN {X 0,Y 192.703,Z 294.108,A -85,B 0,C 180,E1 -21936.348,E2 -21936.348} C_VEL
LIN {X 0,Y 192.729,Z 294.097,A -85,B 0,C 180,E1 -21941.457,E2 -21941.457} C_VEL
LIN {X 0,Y 192.758,Z 294.073,A -85,B 0,C 180,E1 -21945.213,E2 -21945.213} C_VEL
LIN {X 0,Y 192.942,Z 294.058,A -85,B 0,C 180,E1 -21949.566,E2 -21949.566} C_VEL
LIN {X 0,Y 192.981,Z 294.066,A -85,B 0,C 180,E1 -21953.728,E2 -21953.728} C_VEL
LIN {X 0,Y 193.259,Z 294.008,A -85,B 0,C 180,E1 -21957.916,E2 -21957.916} C_VEL
LIN {X 0,Y 193.442,Z 294.005,A -85,B 0,C 180,E1 -21960,E2 -21960} C_VEL
LIN {X 0,Y 192.971,Z 294.043,A -85,B 0,C 180,E1 -21964.177,E2 -21964.177} C_VEL
LIN {X 0,Y 193.064,Z 294.047,A -85,B 0,C 180,E1 -21968.372,E2 -21968.372} C_VEL
LIN {X 0,Y 192.847,Z 294.08,A -85,B 0,C 180,E1 -21972.63,E2 -21972.63} C_VEL
LIN {X 0,Y 192.778,Z 294.088,A -85,B 0,C 180,E1 -21978.586,E2 -21978.586} C_VEL
LIN {X 0,Y 192.661,Z 294.104,A -85,B 0,C 180,E1 -21984.225,E2 -21984.225} C_VEL
LIN {X 0,Y 192.628,Z 294.122,A -85,B 0,C 180,E1 -21989.7,E2 -21989.7} C_VEL
LIN {X 0,Y 192.686,Z 294.542,A -85,B 0,C 180,E1 -21990.706,E2 -21990.706} C_VEL
LIN {X 0,Y 193.239,Z 296.202,A -85,B 0,C 180,E1 -21991.368,E2 -21991.368} C_VEL
LIN {X 0,Y 195.22,Z 298.722,A -85,B 0,C 180,E1 -21992.479,E2 -21992.479} C_VEL
LIN {X 0,Y 196.735,Z 299.854,A -85,B 0,C 180,E1 -21993.239,E2 -21993.239} C_VEL
LIN {X 0,Y 198.614,Z 302.981,A -85,B 0,C 180,E1 -21994.253,E2 -21994.253} C_VEL
LIN {X 0,Y 200.742,Z 305.179,A -85,B 0,C 180,E1 -21995.266,E2 -21995.266} C_VEL
LIN {X 0,Y 203.257,Z 308.724,A -85,B 0,C 180,E1 -21996.462,E2 -21996.462} C_VEL
LIN {X 0,Y 204.777,Z 310.678,A -85,B 0,C 180,E1 -21997.144,E2 -21997.144} C_VEL
LIN {X 0,Y 208.104,Z 315.475,A -85,B 0,C 180,E1 -21998.596,E2 -21998.596} C_VEL
LIN {X 0,Y 214.44,Z 325.912,A -85,B 0,C 180,E1 -22001.189,E2 -22001.189} C_VEL
LIN {X 0,Y 220.264,Z 336.706,A -85,B 0,C 180,E1 -22003.393,E2 -22003.393} C_VEL
LIN {X 0,Y 226.236,Z 349.385,A -85,B 0,C 180,E1 -22005.522,E2 -22005.522} C_VEL
LIN {X 0,Y 228.494,Z 354.773,A -85,B 0,C 180,E1 -22006.305,E2 -22006.305} C_VEL
LIN {X 0,Y 229.037,Z 357.735,A -85,B 0,C 180,E1 -22006.559,E2 -22006.559} C_VEL
LIN {X 0,Y 228.55,Z 362.273,A -85,B 0,C 180,E1 -22006.636,E2 -22006.636} C_VEL
LIN {X 0,Y 225.386,Z 373.702,A -85,B 0,C 180,E1 -22006.367,E2 -22006.367} C_VEL
LIN {X 0,Y 225.111,Z 375.8,A -85,B 0,C 180,E1 -22006.391,E2 -22006.391} C_VEL
LIN {X 0,Y 221.704,Z 430.783,A -85,B 0,C 180,E1 -22008.022,E2 -22008.022} C_VEL
LIN {X 0,Y 219.943,Z 444.554,A -85,B 0,C 180,E1 -22008.698,E2 -22008.698} C_VEL
LIN {X 0,Y 217.618,Z 457.416,A -85,B 0,C 180,E1 -22009.616,E2 -22009.616} C_VEL
LIN {X 0,Y 214.61,Z 470.658,A -85,B 0,C 180,E1 -22010.922,E2 -22010.922} C_VEL
LIN {X 0,Y 211.024,Z 483.423,A -85,B 0,C 180,E1 -22012.57,E2 -22012.57} C_VEL
LIN {X 0,Y 207.543,Z 494.263,A -85,B 0,C 180,E1 -22014.361,E2 -22014.361} C_VEL
LIN {X 0,Y 203.82,Z 504.703,A -85,B 0,C 180,E1 -22016.517,E2 -22016.517} C_VEL
LIN {X 0,Y 199.439,Z 515.417,A -85,B 0,C 180,E1 -22019.273,E2 -22019.273} C_VEL
LIN {X 0,Y 195.611,Z 524.263,A -85,B 0,C 180,E1 -22022.157,E2 -22022.157} C_VEL
LIN {X 0,Y 191.81,Z 532.743,A -85,B 0,C 180,E1 -22025.657,E2 -22025.657} C_VEL
LIN {X 0,Y 189.583,Z 537.763,A -85,B 0,C 180,E1 -22028.241,E2 -22028.241} C_VEL
LIN {X 0,Y 186.672,Z 544.284,A -85,B 0,C 180,E1 -22032.471,E2 -22032.471} C_VEL
LIN {X 0,Y 184.611,Z 549.164,A -85,B 0,C 180,E1 -22036.797,E2 -22036.797} C_VEL
LIN {X 0,Y 183.496,Z 552.557,A -85,B 0,C 180,E1 -22041.188,E2 -22041.188} C_VEL
LIN {X 0,Y 183.018,Z 554.562,A -85,B 0,C 180,E1 -22045.596,E2 -22045.596} C_VEL
LIN {X 0,Y 183.062,Z 555.221,A -85,B 0,C 180,E1 -22050,E2 -22050} C_VEL
LIN {X 0,Y 183.018,Z 554.541,A -85,B 0,C 180,E1 -22054.405,E2 -22054.405} C_VEL
LIN {X 0,Y 183.497,Z 552.519,A -85,B 0,C 180,E1 -22058.812,E2 -22058.812} C_VEL
LIN {X 0,Y 184.614,Z 549.106,A -85,B 0,C 180,E1 -22063.203,E2 -22063.203} C_VEL
LIN {X 0,Y 186.669,Z 544.2,A -85,B 0,C 180,E1 -22067.529,E2 -22067.529} C_VEL
LIN {X 0,Y 189.472,Z 537.655,A -85,B 0,C 180,E1 -22071.772,E2 -22071.772} C_VEL
LIN {X 0,Y 192.794,Z 530.376,A -85,B 0,C 180,E1 -22075.361,E2 -22075.361} C_VEL
LIN {X 0,Y 196.849,Z 521.357,A -85,B 0,C 180,E1 -22078.815,E2 -22078.815} C_VEL
LIN {X 0,Y 200.843,Z 511.895,A -85,B 0,C 180,E1 -22081.66,E2 -22081.66} C_VEL
LIN {X 0,Y 205.025,Z 501.42,A -85,B 0,C 180,E1 -22084.146,E2 -22084.146} C_VEL
LIN {X 0,Y 208.755,Z 490.243,A -85,B 0,C 180,E1 -22086.306,E2 -22086.306} C_VEL
LIN {X 0,Y 212.333,Z 478.604,A -85,B 0,C 180,E1 -22088.058,E2 -22088.058} C_VEL
LIN {X 0,Y 215.507,Z 466.459,A -85,B 0,C 180,E1 -22089.488,E2 -22089.488} C_VEL
LIN {X 0,Y 218.388,Z 453.088,A -85,B 0,C 180,E1 -22090.667,E2 -22090.667} C_VEL
LIN {X 0,Y 220.465,Z 439.391,A -85,B 0,C 180,E1 -22091.563,E2 -22091.563} C_VEL
LIN {X 0,Y 221.875,Z 426.866,A -85,B 0,C 180,E1 -22092.081,E2 -22092.081} C_VEL
LIN {X 0,Y 225.641,Z 364.03,A -85,B 0,C 180,E1 -22093.912,E2 -22093.912} C_VEL
LIN {X 0,Y 225.342,Z 362.315,A -85,B 0,C 180,E1 -22094.06,E2 -22094.06} C_VEL
LIN {X 0,Y 218.718,Z 346.701,A -85,B 0,C 180,E1 -22096.482,E2 -22096.482} C_VEL
LIN {X 0,Y 212.738,Z 334.828,A -85,B 0,C 180,E1 -22098.791,E2 -22098.791} C_VEL
LIN {X 0,Y 207.997,Z 326.331,A -85,B 0,C 180,E1 -22100.752,E2 -22100.752} C_VEL
LIN {X 0,Y 203.271,Z 318.632,A -85,B 0,C 180,E1 -22102.845,E2 -22102.845} C_VEL
LIN {X 0,Y 200.09,Z 314.287,A -85,B 0,C 180,E1 -22104.321,E2 -22104.321} C_VEL
LIN {X 0,Y 197.054,Z 310.178,A -85,B 0,C 180,E1 -22105.825,E2 -22105.825} C_VEL
LIN {X 0,Y 194.407,Z 306.774,A -85,B 0,C 180,E1 -22107.214,E2 -22107.214} C_VEL
LIN {X 0,Y 193.576,Z 305.624,A -85,B 0,C 180,E1 -22107.674,E2 -22107.674} C_VEL
LIN {X 0,Y 191.054,Z 302.898,A -85,B 0,C 180,E1 -22109.08,E2 -22109.08} C_VEL
LIN {X 0,Y 189.836,Z 300.665,A -85,B 0,C 180,E1 -22109.861,E2 -22109.861} C_VEL
LIN {X 0,Y 187.35,Z 298.785,A -85,B 0,C 180,E1 -22111.339,E2 -22111.339} C_VEL
LIN {X 0,Y 185.763,Z 295.993,A -85,B 0,C 180,E1 -22112.543,E2 -22112.543} C_VEL
LIN {X 0,Y 185.558,Z 295.071,A -85,B 0,C 180,E1 -22113.424,E2 -22113.424} C_VEL
LIN {X 0,Y 185.596,Z 294.967,A -85,B 0,C 180,E1 -22117.749,E2 -22117.749} C_VEL
LIN {X 0,Y 185.713,Z 294.955,A -85,B 0,C 180,E1 -22122.377,E2 -22122.377} C_VEL
LIN {X 0,Y 185.761,Z 294.969,A -85,B 0,C 180,E1 -22126.88,E2 -22126.88} C_VEL
LIN {X 0,Y 186.011,Z 294.921,A -85,B 0,C 180,E1 -22131.308,E2 -22131.308} C_VEL
LIN {X 0,Y 186.203,Z 294.898,A -85,B 0,C 180,E1 -22137.837,E2 -22137.837} C_VEL
LIN {X 0,Y 186.403,Z 294.882,A -85,B 0,C 180,E1 -22140,E2 -22140} C_VEL
LIN {X 0,Y 185.916,Z 294.934,A -85,B 0,C 180,E1 -22144.336,E2 -22144.336} C_VEL
LIN {X 0,Y 185.98,Z 294.915,A -85,B 0,C 180,E1 -22148.694,E2 -22148.694} C_VEL
LIN {X 0,Y 185.727,Z 294.96,A -85,B 0,C 180,E1 -22153.123,E2 -22153.123} C_VEL
LIN {X 0,Y 185.687,Z 294.977,A -85,B 0,C 180,E1 -22157.625,E2 -22157.625} C_VEL
LIN {X 0,Y 185.594,Z 294.974,A -85,B 0,C 180,E1 -22162.252,E2 -22162.252} C_VEL
LIN {X 0,Y 185.581,Z 295.194,A -85,B 0,C 180,E1 -22167.029,E2 -22167.029} C_VEL
LIN {X 0,Y 185.857,Z 296.267,A -85,B 0,C 180,E1 -22167.748,E2 -22167.748} C_VEL
